// PLC -> Robot 外圍設備Input(Fanuc Robot的外圍)
MEMMOVE(
destAddr:=ADR(_rawOut_UO[0])
,srcAddr:=ADR(_UI1)
,n:=4
);
// PLC -> Robot Digital Output 2byte(send the command to Fanuc Robot), Warehouse Robot move ClampA
MEMMOVE(
destAddr:=ADR(_rawOut_DO[0])
,srcAddr:=ADR(_DO1)
,n:=2 
);
// PLC -> Robot Digital Output 2byte(send the command to Fanuc Robot), Warehouse Robot move ClampB
MEMMOVE(
destAddr:=ADR(_rawOut_DO[2])
,srcAddr:=ADR(_DO2)
,n:=2 
);
// PLC -> Robot Digital Output 2byte(send the command to Fanuc Robot), ABS Robot move ClampA
MEMMOVE(
destAddr:=ADR(_rawOut_DO[4])
,srcAddr:=ADR(_DO3)
,n:=2 
);
// PLC -> Robot Digital Output 2byte(send the command to Fanuc Robot), ABS Robot move ClampA
MEMMOVE(
destAddr:=ADR(_rawOut_DO[6])
,srcAddr:=ADR(_DO4)
,n:=2 
);
// PLC -> Robot Digital output 2byte(send the command to Fanuc Robot), General Command
MEMMOVE(
destAddr:=ADR(_rawOut_DO[8])
,srcAddr:=ADR(_DO5)
,n:=2 
);
MEMMOVE(
destAddr:=ADR(_rawOut_DO[10])
,srcAddr:=ADR(_DO6)
,n:=2 
);
MEMMOVE(
destAddr:=ADR(_rawOut_DO[12])
,srcAddr:=ADR(_DO7)
,n:=2 
);
MEMMOVE(
destAddr:=ADR(_rawOut_DO[14])
,srcAddr:=ADR(_DO8)
,n:=2 
);
MEMMOVE(
destAddr:=ADR(_rawOut_DO[16])
,srcAddr:=ADR(_DO9)
,n:=2 
);

MEMMOVE(
destAddr:=ADR(_rawOut_DO[18])
,srcAddr:=ADR(_DO10)
,n:=2 
);
MEMMOVE(
destAddr:=ADR(_rawOut_DO[20])
,srcAddr:=ADR(_DO11)
,n:=2 
);
MEMMOVE(
destAddr:=ADR(_rawOut_DO[22])
,srcAddr:=ADR(_DO12)
,n:=2 
);
MEMMOVE(
destAddr:=ADR(_rawOut_DO[24])
,srcAddr:=ADR(_DO13)
,n:=2 
);
MEMMOVE(
destAddr:=ADR(_rawOut_DO[26])
,srcAddr:=ADR(_DO14)
,n:=2 
);
MEMMOVE(
destAddr:=ADR(_rawOut_DO[28])
,srcAddr:=ADR(_DO15)
,n:=2 
);
MEMMOVE(
destAddr:=ADR(_rawOut_DO[30])
,srcAddr:=ADR(_DO16)
,n:=2 
);


// Robot -> PLC Digital Input 3byte(Send Robot Status to PLC), All service
MEMMOVE(
destAddr:=ADR(_DI1)
,srcAddr:=ADR(_rawIn_DI[0])
,n:=3
);

MEMMOVE(
destAddr:=ADR(_DI2)
,srcAddr:=ADR(_rawIn_DI[3])
,n:=2
);
MEMMOVE(
destAddr:=ADR(_DI3)
,srcAddr:=ADR(_rawIn_DI[5])
,n:=2
);
MEMMOVE(
destAddr:=ADR(_DI4)
,srcAddr:=ADR(_rawIn_DI[7])
,n:=2
);
MEMMOVE(
destAddr:=ADR(_DI5)
,srcAddr:=ADR(_rawIn_DI[9])
,n:=2
);
MEMMOVE(
destAddr:=ADR(_DI6)
,srcAddr:=ADR(_rawIn_DI[11])
,n:=2
);
MEMMOVE(
destAddr:=ADR(_DI7)
,srcAddr:=ADR(_rawIn_DI[13])
,n:=2
);
MEMMOVE(
destAddr:=ADR(_DI8)
,srcAddr:=ADR(_rawIn_DI[15])
,n:=2
);
MEMMOVE(
destAddr:=ADR(_DI9)
,srcAddr:=ADR(_rawIn_DI[17])
,n:=2
);
MEMMOVE(
destAddr:=ADR(_DI10)
,srcAddr:=ADR(_rawIn_DI[19])
,n:=2
);
MEMMOVE(
destAddr:=ADR(_DI11)
,srcAddr:=ADR(_rawIn_DI[21])
,n:=2
);
MEMMOVE(
destAddr:=ADR(_DI12)
,srcAddr:=ADR(_rawIn_DI[23])
,n:=2
);

// Robot Status com
qEnable:=_UO1.UO01_CmdEnabled AND _UO1.UO02_SystemReady;
Error:=Fault();

// Velocity Command transfer
_DO5.VelocityBit0 := _VelocityCommand.BitList.Bit0;
_DO5.VelocityBit1 := _VelocityCommand.BitList.Bit1;
_DO5.VelocityBit2 := _VelocityCommand.BitList.Bit2;
_DO5.VelocityBit3 := _VelocityCommand.BitList.Bit3;
_DO5.VelocityBit4 := _VelocityCommand.BitList.Bit4;
_DO5.VelocityBit5 := _VelocityCommand.BitList.Bit5;
_DO5.VelocityBit6 := _VelocityCommand.BitList.Bit6;
_DO5.VelocityBit7 := _VelocityCommand.BitList.Bit7;
END_METHOD

{attribute 'monitoring' := 'variable'}
PROPERTY VelocityCommand : Int
GET
VelocityCommand :=_VelocityCommand.nInt;
END_GET
SET
_VelocityCommand.nInt :=VelocityCommand;
END_SET
END_PROPERTY

PROPERTY WareHouseClampA_Handshake : ST_Fanuc_WarehouseHandshake
GET
WareHouseClampA_Handshake := _DO1;
END_GET
SET
// Outside -> FB 
_DO1 := WareHouseClampA_Handshake;
END_SET
END_PROPERTY

PROPERTY WareHouseClampB_Handshake : ST_Fanuc_WarehouseHandshake
GET
WareHouseClampB_Handshake := _DO2;
END_GET
SET
// Outside -> FB 
_DO2 := WareHouseClampB_Handshake;
END_SET
END_PROPERTY

PROPERTY Write_OffsetP : INT
SET
_DI11 := Write_OffsetP;
END_SET
END_PROPERTY

PROPERTY Write_OffsetR : INT
SET
_DO12 := Write_OffsetR;
END_SET
END_PROPERTY

PROPERTY Write_OffsetW : INT
SET
_DO10 := Write_OffsetW;
END_SET
END_PROPERTY

PROPERTY Write_OffsetX : INT
SET
_DO7 := Write_OffsetX;
END_SET
END_PROPERTY

PROPERTY Write_OffsetY : INT
SET
_DO8 := Write_OffsetY;
END_SET
END_PROPERTY

PROPERTY Write_OffsetZ : INT
SET
_DO9 := Write_OffsetZ;
END_SET
END_PROPERTY

PROPERTY WriteDataCommand : bool;
SET
_DO6.WritePara_Execute := WriteDataCommand;
END_SET
END_PROPERTY

END_FUNCTION_BLOCK

// ---- Library/20_MachineUnits/21_StorageArea/Old_version_Service/FB_FeedInEmptyBoxWithRobot.TcPOU
FUNCTION_BLOCK FB_FeedInEmptyBoxWithRobot EXTENDS FB_ObjectBase_V2 IMPLEMENTS IBasicElement
VAR_INPUT
    // Below are the components being controlled.
    Robot           : REFERENCE TO FB_FanucRobot_Basic_V2; // Fanuc Robot
    PullOutConveyor : REFERENCE TO FB_PullOutConveyorAction; // Allocated area pull out conveyor
    DiffSizeCV  : REFERENCE TO FB_Motor; // Allocated area feed in conveyor(diff and same size conveyor)
	SameSizeCV : REFERENCE TO FB_Motor;
    WareHouse       : REFERENCE TO FB_WareHouse; // Storage area warehouse A and warehouse B conveyor and sensor
    //SameSizeFullSensor : REFERENCE TO BOOL; 				 // Because the same size sensor implement FB_ConveyorSameSize, so use reference to connect it
    Info  : ST_FeedInEmptyBox_Info; // Setting the feedin emptybox action's parameter
    Input : REFERENCE TO ST_InputTable;
    Stop  : BOOL;
END_VAR
VAR_OUTPUT
END_VAR
VAR
    tonPlaceSensorDelay    : TON;
    tonFeedInConveyorDelay : TON;
    tonTimeOut             : TON;
    tonFeedBoxTimeout      : TON;
    strStatus              : STRING;
    _UniqueErrorCode       : STRING;
    _Abort                 : BOOL;
    uiResumeStep           : DINT;
    PreviousStrStatus      : STRING;
    PreviousErrorCode      : STRING;
	
	//2025/11/17 edit by Gamin
	TON_SameSizeCVmove	: TON;
	TON_DiffSizeCVmove	: TON;
END_VAR

SUPER^.A10_StateControl();
A00_BasicUnits();

ACTION A00_BasicUnits:
tonTimeOut(PT:=T#300S);
tonFeedBoxTimeout(PT:=T#15S);
tonPlaceSensorDelay(PT:=T#1S);
tonFeedInConveyorDelay(PT:=T#500MS);

//
TON_SameSizeCVmove(PT :=T#1S);
TON_DiffSizeCVmove(PT :=T#1S);
END_ACTION

METHOD M_CheckCommand : BOOL
VAR_INPUT
END_VAR

VAR_INST
	CheckBehavior : BOOL; // True : Behavior is correct
	CheckWareHouseSetting : BOOL; // True : WareHouse setting is correct
	CheckPullOutConveyorSetting : BOOL; // True : PullOut Conveyor setting is correct
	CheckPickUpArea : BOOL; // True : PickUp Area is correct
	CheckPlaceArea : BOOL; // True : Place Area is correct
END_VAR
// Memory clear
CheckBehavior := FALSE;
// Check command is correct
IF info.ClampA_Setting.Behavior = E_ClampWork.Work OR info.ClampB_Setting.Behavior = E_ClampWork.Work THEN
	CheckBehavior := TRUE;
ELSE
	CheckBehavior := FALSE;
END_IF


M_CheckCommand := CheckBehavior;
END_METHOD

METHOD M_CheckUnitsNotBusy : BOOL
VAR_INPUT
END_VAR
M_CheckUnitsNotBusy := true; // need add units check
END_METHOD

METHOD M_CheckUnitsReady : BOOL
VAR_INPUT
END_VAR
M_CheckUnitsReady := NOT (Robot.Error (*OR PullOutConveyor.Error OR FeedInConveyor.bError OR WareHouse.bError*));
END_METHOD

METHOD M_ReloadBox
VAR_INPUT
	Info : ST_FeedInEmptyBox_Info;
END_VAR
IF info.PickUpArea    = E_FeedInEmptyBox_PickUpArea.PullOutConveyorA THEN
    uiExecutingStep   := 1000;
ELSIF info.PickUpArea = E_FeedInEmptyBox_PickUpArea.PullOutConveyorB THEN
    uiExecutingStep   := 2000;
ELSIF info.PickUpArea = E_FeedInEmptyBox_PickUpArea.WareHouseA THEN
    //WareHouse.
ELSIF info.PickUpArea = E_FeedInEmptyBox_PickUpArea.WareHouseB THEN
    uiExecutingStep   := 4000;
ELSE
    _Error := TRUE;
    Status := 'PickUp area value is out of range';
END_IF
END_METHOD

METHOD M_ReloadPulloutConveyorBox : BOOL
VAR_INPUT
	Execute : BOOL;
	SlideSelect : E_PullOutConveyorPosition;
END_VAR
VAR_INST
	uiReloadPulloutConveyorBoxStep : UDINT;
	fbExecute_Rtrig : R_TRIG;
	fbExecute_Ftrig : F_TRIG;
END_VAR
fbExecute_Rtrig(CLK := Execute);
fbExecute_Ftrig(CLK := Execute);
IF fbExecute_Rtrig.Q THEN
	uiReloadPulloutConveyorBoxStep := 100;
ELSIF fbExecute_Ftrig.Q THEN
	uiReloadPulloutConveyorBoxStep := 99000;
END_IF
CASE uiReloadPulloutConveyorBoxStep OF
	0 : 
		// Wait command
	99000:
//		PullOutConveyor.FixCylinderA1.M_MoveBackward('');
//		PullOutConveyor.FixCylinderA2.M_MoveBackward('');
//		PullOutConveyor.FixCylinderB1.M_MoveBackward('');
//		PullOutConveyor.FixCylinderB2.M_MoveBackward('');
END_CASE
END_METHOD

METHOD M_SelectActionMode : E_FeedInAction
VAR_INPUT
END_VAR
IF info.ClampA_Setting.Behavior = E_ClampWork.Work AND info.ClampB_Setting.Behavior <> E_ClampWork.Work THEN
	IF info.ClampA_Setting.PickUpArea = E_FeedInEmptyBox_PickUpArea.WareHouseA THEN
		M_SelectActionMode := E_FeedInAction.ClampA_WareHouseA;
	ELSIF info.ClampA_Setting.PickUpArea = E_FeedInEmptyBox_PickUpArea.WareHouseB THEN
		M_SelectActionMode := E_FeedInAction.ClampA_WareHouseB;
	ELSIF info.ClampA_Setting.PickUpArea = E_FeedInEmptyBox_PickUpArea.PullOutConveyor THEN
		M_SelectActionMode := E_FeedInAction.ClampA_PullOutConveyor;
	END_IF
ELSIF info.ClampA_Setting.Behavior <> E_ClampWork.Work AND info.ClampB_Setting.Behavior = E_ClampWork.Work THEN
	IF info.ClampB_Setting.PickUpArea = E_FeedInEmptyBox_PickUpArea.WareHouseA THEN
		M_SelectActionMode := E_FeedInAction.ClampB_WareHouseA;
	ELSIF info.ClampB_Setting.PickUpArea = E_FeedInEmptyBox_PickUpArea.WareHouseB THEN
		M_SelectActionMode := E_FeedInAction.ClampB_WareHouseB;
	ELSIF info.ClampB_Setting.PickUpArea = E_FeedInEmptyBox_PickUpArea.PullOutConveyor THEN
		M_SelectActionMode := E_FeedInAction.ClampB_PullOutConveyor;
	END_IF
ELSIF info.ClampA_Setting.Behavior = E_ClampWork.Work AND info.ClampB_Setting.Behavior = E_ClampWork.Work THEN
	IF info.ClampA_Setting.PickUpArea = E_FeedInEmptyBox_PickUpArea.PullOutConveyor THEN
		IF  info.ClampB_Setting.PickUpArea = E_FeedInEmptyBox_PickUpArea.WareHouseA THEN
			M_SelectActionMode := E_FeedInAction.A_PullOut_B_WareHouseA;
		ELSIF info.ClampB_Setting.PickUpArea = E_FeedInEmptyBox_PickUpArea.WareHouseB THEN
			M_SelectActionMode := E_FeedInAction.A_PullOut_B_WareHouseB;
		ELSIF info.ClampB_Setting.PickUpArea = E_FeedInEmptyBox_PickUpArea.PullOutConveyor THEN
			M_SelectActionMode := E_FeedInAction.A_PullOut_B_PullOut;
		END_IF
	ELSIF info.ClampA_Setting.PickUpArea = E_FeedInEmptyBox_PickUpArea.WareHouseA THEN
		IF info.ClampB_Setting.PickUpArea = E_FeedInEmptyBox_PickUpArea.WareHouseA THEN
			M_SelectActionMode := E_FeedInAction.A_WareHouseA_B_WareHouseA;
		ELSIF info.ClampB_Setting.PickUpArea = E_FeedInEmptyBox_PickUpArea.WareHouseB THEN
			M_SelectActionMode := E_FeedInAction.A_WareHouseA_B_WareHouseB;
		ELSIF info.ClampB_Setting.PickUpArea = E_FeedInEmptyBox_PickUpArea.PullOutConveyor THEN
			M_SelectActionMode := E_FeedInAction.A_WareHouseA_B_PullOut;
		END_IF
	ELSIF info.ClampA_Setting.PickUpArea = E_FeedInEmptyBox_PickUpArea.WareHouseB THEN
		IF info.ClampB_Setting.PickUpArea = E_FeedInEmptyBox_PickUpArea.WareHouseA THEN
			M_SelectActionMode := E_FeedInAction.A_WareHouseB_B_WareHouseA;
		ELSIF info.ClampB_Setting.PickUpArea = E_FeedInEmptyBox_PickUpArea.WareHouseB THEN
			M_SelectActionMode := E_FeedInAction.A_WareHouseB_B_WareHouseB;
		ELSIF info.ClampB_Setting.PickUpArea = E_FeedInEmptyBox_PickUpArea.PullOutConveyor THEN
			M_SelectActionMode := E_FeedInAction.A_WareHouseB_B_PullOut;
		END_IF
	END_IF
END_IF
END_METHOD

METHOD  M_STATE_ABORTED
VAR_INPUT
END_VAR
Busy    := FALSE;
Aborted := TRUE;
Status := strStatus ;
UniqueErrorCode := _UniqueErrorCode;
IF NOT Execute THEN
    eState := STATE_RESETTING;
END_IF

IF Execute AND Reset THEN
	uiExecutingStep :=uiResumeStep;
	PreviousStrStatus := strStatus;
	PreviousErrorCode := _UniqueErrorCode;
	eState :=STATE_EXECUTING;
END_IF
END_METHOD

METHOD  M_STATE_ABORTING
VAR_INPUT
END_VAR
_AbortCompleted := TRUE;
_Abort :=FALSE;
tonTimeOut.IN:=FALSE;
//DAS.fbStorageArea.M_ResetSlideA_FeedIn();
IF strStatus = PreviousStrStatus THEN
	_UniqueErrorCode :=PreviousErrorCode;
END_IF
IF _AbortCompleted THEN
    eState := STATE_Aborted;
END_IF
END_METHOD

METHOD  M_STATE_DONE
VAR_INPUT
END_VAR
Busy := FALSE;
Done := TRUE;
IF NOT Execute THEN
    eState := STATE_RESETTING;
END_IF
END_METHOD

METHOD  M_STATE_DORMANT
VAR_INPUT
END_VAR
// Clear FB output
Busy            := FALSE;
Done            := FALSE;
Aborted         := FALSE;
Error           :=  FALSE;
ErrorID         := 0;
Status          := '';
_ResetCompleted := FALSE;
_Error          := FALSE;
_Executed       := FALSE;
uiExecutingStep := 0;
uiResettingStep := 0;
uiResumeStep:=0;
tonPlaceSensorDelay.IN :=FALSE;
tonFeedInConveyorDelay.IN :=FALSE;
tonTimeOut.IN :=FALSE;
TON_DiffSizeCVmove.IN := FALSE;
TON_SameSizeCVmove.IN := FALSE;
_UniqueErrorCode :='0';
PreviousStrStatus			 :='';
PreviousErrorCode			 :='';
//DAS.fbStorageArea.M_InactivePulloutConveyorInternCtrl();
// Wait Execute command
IF Execute THEN
    eState := STATE_EXECUTING;
END_IF
END_METHOD

METHOD  M_STATE_ERROR
VAR_INPUT
END_VAR
Robot.Bzone_AllowWork:=FALSE;
IF NOT Execute THEN
    eState := STATE_RESETTING;
END_IF
END_METHOD

METHOD M_STATE_EXECUTING
VAR_INPUT
END_VAR
VAR_INST
    ClampA_WareHouseCoordinates : ST_WareHouseCoordinates;
    ClampB_WareHouseCoordinates : ST_WareHouseCoordinates;
    uiPickUpBothStep            : UINT;
    uiPlaceBothStep             : UINT;
    BoxReady_1st                : BOOL;
    BoxReady_2nd                : BOOL;
    SlideClear_1st              : BOOL;
    SlideClear_2nd              : BOOL;
    TargetWarehouse             : E_WareHouse;
    DiffSizeSlide_Clear         : BOOL;
    SameSizeSlide_clear         : BOOL;
    ActionMode                  : E_FeedInAction;
END_VAR
VAR

END_VAR
// Set status busy
Busy := TRUE;
Robot.Bzone_AllowWork:=Robot._DI12.BzoneInWork;
//Auto mode , just allow robot
IF THIS^.Stop THEN // Pending the timeout when Stop signal occur
  tonTimeout.IN :=FALSE;
END_IF
CASE uiExecutingStep OF
    0:
        // Clear variable
        ActionMode       := E_FeedInAction.Undefined;
        BoxReady_1st     := FALSE;
        BoxReady_2nd     := FALSE;
        uiPickUpBothStep := 0;
        uiPlaceBothStep  := 0;

        // Check command
        IF M_CheckCommand() THEN
            uiExecutingStep := 10;
        END_IF
    10: // Start process, check units first
        IF M_CheckUnitsReady() THEN
            uiExecutingStep := 20;
        END_IF
    20: // Check units not busy state
        IF M_CheckUnitsNotBusy() THEN
            uiExecutingStep := 1000;
        END_IF
    1000:
        // Select action mode
        ActionMode      := M_SelectActionMode();
        uiExecutingStep := 1100;
    1100:
        // according action mode jump step
        CASE ActionMode OF
            E_FeedInAction.ClampA_WareHouseA:
                uiExecutingStep := 10000; // Go to start only ClampA pickup from WareHouseA
            E_FeedInAction.ClampA_WareHouseB:
                uiExecutingStep := 11000; // Go to Start only ClampA pickup from WareHouseB
            E_FeedInAction.ClampA_PullOutConveyor:
                uiExecutingStep := 12000; // Go to Start only ClampA pickup form PulloutConveyor
            E_FeedInAction.ClampB_WareHouseA:
                uiExecutingStep := 20000; // Go to Start only ClampB pickup from WareHouseA
            E_FeedInAction.ClampB_WareHouseB:
                uiExecutingStep := 21000; // Go to Start only ClampB pickup from WareHouseB
            E_FeedInAction.ClampB_PullOutConveyor:
                uiExecutingStep := 22000; // Go to Start only ClampB pickup from PulloutConveyor
            E_FeedInAction.A_WareHouseA_B_WareHouseA:
                uiExecutingStep := 30000; // Go to Start ClampA pickup from WarehouseA, ClampB pickup from WarehouseA
            E_FeedInAction.A_WareHouseA_B_WareHouseB:
                uiExecutingStep := 31000; // Go to Start ClampA pickup from WarehouseA, ClmapB pickup from WarehouseB
            E_FeedInAction.A_WareHouseA_B_PullOut:
                uiExecutingStep := 32000; // Go to Start ClampA pickup from WarehouseA, ClampB pickup from PulloutConveyor
            E_FeedInAction.A_WareHouseB_B_WareHouseA:
                uiExecutingStep := 33000; // Go to Start ClampA pickup from WarehouseB, ClampB pickup from WarehouseA
            E_FeedInAction.A_WareHouseB_B_WareHouseB:
                uiExecutingStep := 34000; // Go to Start ClampA pickup from WarehouseB, CLampB pickup from WarehouseB
            E_FeedInAction.A_WareHouseB_B_PullOut:
                uiExecutingStep := 35000; // Go to Start ClampA pickup from WarehouseB, ClampB pickup from PulloutConveyor
            E_FeedInAction.A_PullOut_B_WareHouseA:
                uiExecutingStep := 36000; // Go to Start ClampA pickup from PulloutConveyor, ClampB pickup from WarehouseA
            E_FeedInAction.A_PullOut_B_WareHouseB:
                uiExecutingStep := 37000; // Go to Start ClampA pickup from PulloutConveyor, ClampB pickup from WarehouseB
            E_FeedInAction.A_PullOut_B_PullOut:
                uiExecutingStep := 38000; // Go to Start ClampBoth pickup from PulloutConveyor
        END_CASE
    10000: // Only clampA pickup box from WareHouseA
        IF NOT Robot._DI1.Done THEN
            ClampA_WareHouseCoordinates := info.ClampA_Setting.WareHouseSetting;
            WareHouse.M_StartReloadBox(WareHouseSelect := E_WareHouse.WareHouseA, WarehouseCoordinates := ClampA_WareHouseCoordinates);

            IF WareHouse.bReloadBox_Completed THEN
                BoxReady_1st := TRUE;
            END_IF

            Robot.M_StartWareHousePickUpBox_ClampA(WareHouseSelect := E_WareHouse.WareHouseA,
                                                   Info            := ClampA_WareHouseCoordinates,
                                                   BoxReady_1st    := BoxReady_1st);
        ELSE
            IF Robot.M_ResetWareHousePickUpBox_ClampA() THEN
                // Clear command and go to place box
        tonTimeOut.IN:=FALSE;
                uiExecutingStep := 60000; // only place clampA
            END_IF
        END_IF
    tonTimeOut.IN :=TRUE;   
    IF tonTimeOut.Q THEN
      tonTimeOut.IN:=FALSE;
      _Error :=TRUE;
      strStatus :='Pick Box timeout';
    END_IF
    
    11000: // Only ClampA pickup box from WareHouseB
        IF NOT Robot._di1.Done THEN
            ClampA_WareHouseCoordinates := info.ClampA_Setting.WareHouseSetting;
            WareHouse.M_StartReloadBox(WareHouseSelect := E_WareHouse.WareHouseB, WarehouseCoordinates := ClampA_WareHouseCoordinates);

            IF WareHouse.bReloadBox_Completed THEN
                BoxReady_1st := TRUE;
            END_IF

            Robot.M_StartWareHousePickUpBox_ClampA(WareHouseSelect := E_WareHouse.WareHouseB,
                                                   Info            := ClampA_WareHouseCoordinates,
                                                   BoxReady_1st    := BoxReady_1st);
        ELSE
            IF Robot.M_ResetWareHousePickUpBox_ClampA() THEN
                // Clear command and go to place box
        tonTimeOut.IN:=FALSE;
                uiExecutingStep := 60000; // only place clampA
            END_IF
        END_IF

    tonTimeOut.IN :=TRUE;   
    IF tonTimeOut.Q THEN
      tonTimeOut.IN:=FALSE;
      _Error :=TRUE;
      strStatus :='Pick Box timeout';
    END_IF
    
    12000: // Only ClampA pickup box from pullout conveyor
        IF NOT Robot._di1.Done THEN
            DAS_CoreSys.MachineControl.fbStorageArea.M_ActivePulloutConveyorInternCtrl();

            IF Info.ClampA_Setting.PullOutConveyorSetting = E_PullOutConveyorAddress.I3_Slide THEN
                DAS_CoreSys.MachineControl.fbStorageArea.M_StartSlideB_FeedIn();
            ELSIF Info.ClampA_Setting.PullOutConveyorSetting = E_PullOutConveyorAddress.I4_Slide THEN
                DAS_CoreSys.MachineControl.fbStorageArea.M_StartSlideA_FeedIn();
            ELSE
                Status := 'Not define PulloutConveyor Slide';
                _Error := TRUE;
            END_IF

            Robot.M_StartPullOutConveyorPickUpBox_ClampA(ClampA_Address := Info.ClampA_Setting.PullOutConveyorSetting,
                                                         BoxReady       := DAS_CoreSys.MachineControl.fballocatearea.fbPulloutCV.Done);
        ELSE
            IF Robot.M_ResetPullOutConveyorPickUpBox_ClampA() THEN
                DAS_CoreSys.MachineControl.fbStorageArea.M_ResetSlideA_FeedIn();
        tonTimeOut.IN:=FALSE;
                uiExecutingStep := 60000; // only place clampA
            END_IF
        END_IF;
      tonTimeOut.IN :=TRUE;   
    IF tonTimeOut.Q THEN
      tonTimeOut.IN:=FALSE;
      _Abort :=TRUE;
      uiResumeStep:=12000;
      strStatus :='Pick Box timeout';
    END_IF
    
    20000: // Only clampB pickup box from WareHouseA
        IF NOT Robot._di1.Done THEN
            ClampB_WareHouseCoordinates := info.ClampB_Setting.WareHouseSetting;
            WareHouse.M_StartReloadBox(WareHouseSelect := E_WareHouse.WareHouseA, WarehouseCoordinates := ClampB_WareHouseCoordinates);

            IF WareHouse.bReloadBox_Completed THEN
                BoxReady_2nd := TRUE;
            END_IF

            Robot.M_StartWareHousePickUpBox_ClampB(WareHouseSelect := E_WareHouse.WareHouseA,
                                                   Info            := ClampB_WareHouseCoordinates,
                                                   BoxReady_2nd    := BoxReady_2nd);
        ELSE
            IF Robot.M_ResetWareHousePickUpBox_ClampB() THEN
                // Clear command and go to place box
        tonTimeOut.IN:=FALSE;
                uiExecutingStep := 70000; // only place clampA
            END_IF
        END_IF
      tonTimeOut.IN :=TRUE;   
    IF tonTimeOut.Q THEN
      tonTimeOut.IN:=FALSE;
      _Error :=TRUE;
      strStatus :='Pick Box timeout';
    END_IF
    21000: // Only ClampB pickup box from WareHouseB
        IF NOT Robot._di1.Done THEN
            ClampB_WareHouseCoordinates := info.ClampB_Setting.WareHouseSetting;
            WareHouse.M_StartReloadBox(WareHouseSelect := E_WareHouse.WareHouseB, WarehouseCoordinates := ClampB_WareHouseCoordinates);

            IF WareHouse.bReloadBox_Completed THEN
                BoxReady_2nd := TRUE;
            END_IF

            Robot.M_StartWareHousePickUpBox_ClampB(WareHouseSelect := E_WareHouse.WareHouseB,
                                                   Info            := ClampB_WareHouseCoordinates,
                                                   BoxReady_2nd    := BoxReady_2nd);
        ELSE
            IF Robot.M_ResetWareHousePickUpBox_ClampB() THEN
                // Clear command and go to place box
        tonTimeOut.IN:=FALSE;
                uiExecutingStep := 70000; // only place clampA
            END_IF
        END_IF
        tonTimeOut.IN :=TRUE;   
    IF tonTimeOut.Q THEN
      tonTimeOut.IN:=FALSE;
      _Error :=TRUE;
      strStatus :='Pick Box timeout';
    END_IF

    22000: // Only ClampB pickup box from PullOut conveyor
        IF NOT Robot._di1.Done THEN
            DAS_CoreSys.MachineControl.fbStorageArea.M_ActivePulloutConveyorInternCtrl();

            IF Info.ClampB_Setting.PullOutConveyorSetting = E_PullOutConveyorAddress.I3_Slide THEN
                DAS_CoreSys.MachineControl.fbStorageArea.M_StartSlideB_FeedIn();
            ELSIF Info.ClampB_Setting.PullOutConveyorSetting = E_PullOutConveyorAddress.I4_Slide THEN
                DAS_CoreSys.MachineControl.fbStorageArea.M_StartSlideA_FeedIn();
            ELSE
                Status := 'Not define PulloutConveyor Slide';
                _Error := TRUE;
            END_IF

            Robot.M_StartPullOutConveyorPickUpBox_ClampB(ClampB_Address := Info.ClampB_Setting.PullOutConveyorSetting,
                                                         BoxReady       := DAS_CoreSys.MachineControl.fballocatearea.fbPulloutCV.Done);
        ELSE
            IF Robot.M_ResetPullOutConveyorPickUpBox_ClampB() THEN
                DAS_CoreSys.MachineControl.fbStorageArea.M_ResetSlideA_FeedIn();
        tonTimeOut.IN:=FALSE;
                uiExecutingStep := 70000; // only place clampA
            END_IF
        END_IF;
      tonTimeOut.IN :=TRUE;   
    IF tonTimeOut.Q THEN
      uiResumeStep:=22000;
      _Abort :=TRUE;
      strStatus :='Pick Box timeout';
    END_IF
    
    30000: // ClampA pickup from WarehouseA, ClampB pickup from WarehouseA
        ClampA_WareHouseCoordinates := info.ClampA_Setting.WareHouseSetting;
        ClampB_WareHouseCoordinates := info.ClampB_Setting.WareHouseSetting;

        CASE uiPickUpBothStep OF
            0: // ClampA target slide move the box to front side
                WareHouse.M_StartReloadBox(WareHouseSelect := E_WareHouse.WareHouseA, WarehouseCoordinates := ClampA_WareHouseCoordinates);

                IF WareHouse.bReloadBox_Completed THEN
                    BoxReady_1st     := TRUE;
                    uiPickUpBothStep := 10;
                END_IF

            10: // wait Robot Allow continue
                IF Robot._DI1.Notification AND
                    NOT
                    WareHouse._stWarehouseList.ASide_Layers[ClampA_WareHouseCoordinates.Layer].stStatus.bSlides[ClampA_WareHouseCoordinates.Slide]
                    THEN
                    WareHouse.M_ResetReloadBox();

                    IF NOT WareHouse.bReloadBox_Completed THEN
                        uiPickUpBothStep := 20;
                    END_IF

                END_IF
            20: // ClampB target slide move the box to front slide
                WareHouse.M_StartReloadBox(WareHouseSelect := E_WareHouse.WareHouseA, WarehouseCoordinates := ClampB_WareHouseCoordinates);

                IF WareHouse.bReloadBox_Completed THEN
                    BoxReady_2nd     := TRUE;
                    uiPickUpBothStep := 99;
                END_IF
            99:
        // wait reset
        END_CASE

        Robot.M_StartWareHousePickUpBox_ClampBoth(WareHouseSelect := E_WareHouse.WareHouseA,
                                                  ClampA_Info     := ClampA_WareHouseCoordinates,
                                                  ClampB_Info     := ClampB_WareHouseCoordinates,
                                                  BoxReady_1st    := BoxReady_1st,
                                                  BoxReady_2nd    := BoxReady_2nd);

        IF Robot._DI1.Done THEN
      tonTimeOut.IN:=FALSE;
            uiExecutingStep := 80000; // go to place step
        END_IF
      tonTimeOut.IN :=TRUE;   
    IF tonTimeOut.Q THEN
      tonTimeOut.IN:=FALSE;
      _Error :=TRUE;
      strStatus :='Pick Box timeout';
    END_IF
    
    31000: // ClampA pickup from WarehouseA, ClampB pickup from WarehouseB
        IF NOT Robot._DI1.Done THEN
            ClampA_WareHouseCoordinates := info.ClampA_Setting.WareHouseSetting;
            WareHouse.M_StartReloadBox(WareHouseSelect := E_WareHouse.WareHouseA, WarehouseCoordinates := ClampA_WareHouseCoordinates);

            IF WareHouse.bReloadBox_Completed THEN
                BoxReady_1st := TRUE;
            END_IF

            Robot.M_StartWareHousePickUpBox_ClampA(WareHouseSelect := E_WareHouse.WareHouseA,
                                                   Info            := ClampA_WareHouseCoordinates,
                                                   BoxReady_1st    := BoxReady_1st);
        ELSE
      tonTimeOut.IN:=FALSE;
      uiExecutingStep := 31080;
    END_IF
      tonTimeOut.IN :=TRUE;   
    IF tonTimeOut.Q THEN
      tonTimeOut.IN:=FALSE;
      _Error :=TRUE;
      strStatus :='Pick Box timeout';
    END_IF
    
  31080:
    Robot.M_ResetAllCommand(); // Clear command and go to place box
    IF NOT Robot._di1.Done THEN
      uiExecutingStep := 31100;// ClampA pickup finished, ClampB pickup start
    END_IF
    
    31100:
        IF NOT Robot._di1.Done THEN
            ClampB_WareHouseCoordinates := info.ClampB_Setting.WareHouseSetting;
            WareHouse.M_StartReloadBox(WareHouseSelect := E_WareHouse.WareHouseB, WarehouseCoordinates := ClampB_WareHouseCoordinates);

            IF WareHouse.bReloadBox_Completed THEN
                BoxReady_2nd := TRUE;
            END_IF

            Robot.M_StartWareHousePickUpBox_ClampB(WareHouseSelect := E_WareHouse.WareHouseB,
                                                   Info            := ClampB_WareHouseCoordinates,
                                                   BoxReady_2nd    := BoxReady_2nd);
        ELSE
      tonTimeOut.IN:=FALSE;
      uiExecutingStep := 31180;
    END_IF
      tonTimeOut.IN :=TRUE;   
    IF tonTimeOut.Q THEN
      tonTimeOut.IN:=FALSE;
      _Error :=TRUE;
      strStatus :='Pick Box timeout';
    END_IF
    
  31180:
    Robot.M_ResetAllCommand(); // Clear command and go to place box
    IF NOT Robot._di1.Done THEN
      uiExecutingStep := 80000;// ClampA pickup finished, ClampB pickup start
    END_IF
    32000: // ClampA pickup from WarehouseA, ClampB pickup from PulloutConveyor
        IF NOT Robot._DI1.Done THEN
            ClampA_WareHouseCoordinates := info.ClampA_Setting.WareHouseSetting;
            WareHouse.M_StartReloadBox(WareHouseSelect := E_WareHouse.WareHouseA, WarehouseCoordinates := ClampA_WareHouseCoordinates);

            IF WareHouse.bReloadBox_Completed THEN
                BoxReady_1st := TRUE;
            END_IF

            Robot.M_StartWareHousePickUpBox_ClampA(WareHouseSelect := E_WareHouse.WareHouseA,
                                                   Info            := ClampA_WareHouseCoordinates,
                                                   BoxReady_1st    := BoxReady_1st);
        ELSE
      tonTimeOut.IN:=FALSE;
      uiExecutingStep := 32080; // ClampA pickup finished, ClampB start 
        END_IF
      tonTimeOut.IN :=TRUE;   
    IF tonTimeOut.Q THEN
      tonTimeOut.IN:=FALSE;
      _Error :=TRUE;
      strStatus :='Pick Box timeout';
    END_IF
  32080:
    Robot.M_ResetAllCommand();
    // Clear command and go to place box
    IF NOT Robot._di1.Done THEN
      uiExecutingStep := 32100;// ClampA pickup finished, ClampB start
    END_IF
    32100:
        IF NOT Robot._di1.Done THEN
        DAS_CoreSys.MachineControl.fballocatearea.M_GetPulloutAccess(ControlAccess := E_RoundBeltControlAccess.FanucRobot);

            IF Info.ClampB_Setting.PullOutConveyorSetting = E_PullOutConveyorAddress.I3_Slide THEN
                        DAS_CoreSys.MachineControl.fballocatearea
                            .M_StartStoragePulloutAction(CommandType := E_PullOutConveyorCommandType.SlideB_FeedIn_Ext,
                                                         CV_BackwardTIme := T#0S,
                                                         CV_ForwardTime := T#0S);
            ELSIF Info.ClampB_Setting.PullOutConveyorSetting = E_PullOutConveyorAddress.I4_Slide THEN
                        DAS_CoreSys.MachineControl.fballocatearea
                            .M_StartStoragePulloutAction(CommandType := E_PullOutConveyorCommandType.SlideA_FeedIn_Ext,
                                                         CV_BackwardTIme := T#0S,
                                                         CV_ForwardTime := T#0S);
            ELSE
                Status := 'Not define PulloutConveyor Slide';
                _Error := TRUE;
            END_IF

            Robot.M_StartPullOutConveyorPickUpBox_ClampB(ClampB_Address := Info.ClampB_Setting.PullOutConveyorSetting,
                                                         BoxReady       := DAS_CoreSys.MachineControl.fballocatearea.fbPulloutCV.Done);
        ELSE
      tonTimeOut.IN:=FALSE;
      uiExecutingStep := 32180;
    END_IF
      tonTimeOut.IN :=TRUE;   
    IF tonTimeOut.Q THEN
      tonTimeOut.IN:=FALSE;
      _Error :=TRUE;
      strStatus :='Pick Box timeout';
    END_IF
  32180:
    robot.M_ResetAllCommand();
    IF NOT Robot._DI1.Done THEN
      uiExecutingStep := 80000;
    END_IF
    33000: // ClampA Pickup from WarehouseB, ClampB pickup from WarehouseA
        IF NOT Robot._di1.Done THEN
            ClampA_WareHouseCoordinates := info.ClampA_Setting.WareHouseSetting;
            WareHouse.M_StartReloadBox(WareHouseSelect := E_WareHouse.WareHouseB, WarehouseCoordinates := ClampA_WareHouseCoordinates);

            IF WareHouse.bReloadBox_Completed THEN
                BoxReady_1st := TRUE;
            END_IF

            Robot.M_StartWareHousePickUpBox_ClampA(WareHouseSelect := E_WareHouse.WareHouseB,
                                                   Info            := ClampA_WareHouseCoordinates,
                                                   BoxReady_1st    := BoxReady_1st);
        ELSE
      tonTimeOut.IN:=FALSE;
      uiExecutingStep := 33080;
    END_IF
        tonTimeOut.IN :=TRUE;   
    IF tonTimeOut.Q THEN
      tonTimeOut.IN:=FALSE;
      _Error :=TRUE;
      strStatus :='Pick Box timeout';
    END_IF
  33080:
    Robot.M_ResetAllCommand(); // Clear command and go to place box
    IF NOT Robot._DI1.Done THEN
                uiExecutingStep := 33100; // only place clampA
        END_IF
    33100:
        IF NOT Robot._di1.Done THEN
            ClampB_WareHouseCoordinates := info.ClampB_Setting.WareHouseSetting;
            WareHouse.M_StartReloadBox(WareHouseSelect := E_WareHouse.WareHouseA, WarehouseCoordinates := ClampB_WareHouseCoordinates);

            IF WareHouse.bReloadBox_Completed THEN
                BoxReady_2nd := TRUE;
            END_IF

            Robot.M_StartWareHousePickUpBox_ClampB(WareHouseSelect := E_WareHouse.WareHouseA,
                                                   Info            := ClampB_WareHouseCoordinates,
                                                   BoxReady_2nd    := BoxReady_2nd);
        ELSE
      Robot.M_ResetAllCommand(); // Clear command and go to place box
      IF NOT Robot._DI1.Done THEN
        tonTimeOut.IN:=FALSE;
        uiExecutingStep := 80000; // only place clampA
      END_IF
        END_IF
    tonTimeOut.IN :=TRUE;   
    IF tonTimeOut.Q THEN
      tonTimeOut.IN:=FALSE;
      _Error :=TRUE;
      strStatus :='Place Box timeout';
    END_IF
    
    34000: // ClampA pickup from WarehouseB, ClampB pickup from WarehouseB
        ClampA_WareHouseCoordinates := info.ClampA_Setting.WareHouseSetting;
        ClampB_WareHouseCoordinates := info.ClampB_Setting.WareHouseSetting;

        CASE uiPickUpBothStep OF
            0: // ClampA target slide move the box to front side
                WareHouse.M_StartReloadBox(WareHouseSelect := E_WareHouse.WareHouseB, WarehouseCoordinates := ClampA_WareHouseCoordinates);

                IF WareHouse.bReloadBox_Completed THEN
                    BoxReady_1st     := TRUE;
                    uiPickUpBothStep := 10;
                END_IF

            10: // wait Robot Allow continue
                IF Robot._DI1.Notification AND
                    NOT
                    WareHouse._stWarehouseList.BSide_Layers[ClampA_WareHouseCoordinates.Layer].stStatus.bSlides[ClampA_WareHouseCoordinates.Slide]
                    THEN
                    WareHouse.M_ResetReloadBox();

                    IF NOT WareHouse.bReloadBox_Completed THEN
                        uiPickUpBothStep := 20;
                    END_IF

                END_IF
            20: // ClampB target slide move the box to front slide
                WareHouse.M_StartReloadBox(WareHouseSelect := E_WareHouse.WareHouseB, WarehouseCoordinates := ClampB_WareHouseCoordinates);

                IF WareHouse.bReloadBox_Completed THEN
                    BoxReady_2nd     := TRUE;
                    uiPickUpBothStep := 99;
                END_IF
            99:
        // wait reset
        END_CASE

        Robot.M_StartWareHousePickUpBox_ClampBoth(WareHouseSelect := E_WareHouse.WareHouseB,
                                                  ClampA_Info     := ClampA_WareHouseCoordinates,
                                                  ClampB_Info     := ClampB_WareHouseCoordinates,
                                                  BoxReady_1st    := BoxReady_1st,
                                                  BoxReady_2nd    := BoxReady_2nd);

        IF Robot._DI1.Done THEN
      tonTimeOut.IN:=FALSE;
            uiExecutingStep := 80000; // go to place step
        END_IF
    
      tonTimeOut.IN :=TRUE;   
    IF tonTimeOut.Q THEN
      tonTimeOut.IN:=FALSE;
      _Error :=TRUE;
      strStatus :='Pick Box timeout';
    END_IF
    
    35000: // ClampA pickup from WarehouseB, ClampB pickup from PulloutConveyor
        IF NOT Robot._di1.Done THEN
        DAS_CoreSys.MachineControl.fballocatearea.M_GetPulloutAccess(ControlAccess := E_RoundBeltControlAccess.FanucRobot);

            IF Info.ClampA_Setting.PullOutConveyorSetting = E_PullOutConveyorAddress.I3_Slide THEN
                        DAS_CoreSys.MachineControl.fballocatearea
                            .M_StartStoragePulloutAction(CommandType := E_PullOutConveyorCommandType.SlideB_FeedIn_Ext,
                                                         CV_BackwardTIme := T#0S,
                                                         CV_ForwardTime := T#0S);
            ELSIF Info.ClampA_Setting.PullOutConveyorSetting = E_PullOutConveyorAddress.I4_Slide THEN
                        DAS_CoreSys.MachineControl.fballocatearea
                            .M_StartStoragePulloutAction(CommandType := E_PullOutConveyorCommandType.SlideA_FeedIn_Ext,
                                                         CV_BackwardTIme := T#0S,
                                                         CV_ForwardTime := T#0S);
            ELSE
                Status := 'Not define PulloutConveyor Slide';
                _Error := TRUE;
            END_IF

            Robot.M_StartPullOutConveyorPickUpBox_ClampA(ClampA_Address := Info.ClampA_Setting.PullOutConveyorSetting,
                                                         BoxReady       := DAS_CoreSys.MachineControl.fballocatearea.fbPulloutCV.Done);
        ELSE
            IF Robot.M_ResetPullOutConveyorPickUpBox_ClampA() THEN
            DAS_CoreSys.MachineControl.fballocatearea.M_StopStoragePulloutAction();
        tonTimeOut.IN:=FALSE;
                uiExecutingStep := 35100; // only place clampA
            END_IF
        END_IF;
      tonTimeOut.IN :=TRUE;   
    IF tonTimeOut.Q THEN
      tonTimeOut.IN:=FALSE;
      _Error :=TRUE;
      strStatus :='Pick Box timeout';
    END_IF
    
    35100:
        IF NOT Robot._di1.Done THEN
        DAS_CoreSys.MachineControl.fballocatearea.M_GetPulloutAccess(ControlAccess := E_RoundBeltControlAccess.FanucRobot);

            IF Info.ClampB_Setting.PullOutConveyorSetting = E_PullOutConveyorAddress.I3_Slide THEN
                        DAS_CoreSys.MachineControl.fballocatearea
                            .M_StartStoragePulloutAction(CommandType := E_PullOutConveyorCommandType.SlideB_FeedIn_Ext,
                                                         CV_BackwardTIme := T#0S,
                                                         CV_ForwardTime := T#0S);
            ELSIF Info.ClampB_Setting.PullOutConveyorSetting = E_PullOutConveyorAddress.I4_Slide THEN
                        DAS_CoreSys.MachineControl.fballocatearea
                            .M_StartStoragePulloutAction(CommandType := E_PullOutConveyorCommandType.SlideA_FeedIn_Ext,
                                                         CV_BackwardTIme := T#0S,
                                                         CV_ForwardTime := T#0S);
            ELSE
                Status := 'Not define PulloutConveyor Slide';
                _Error := TRUE;
            END_IF

            Robot.M_StartPullOutConveyorPickUpBox_ClampB(ClampB_Address := Info.ClampB_Setting.PullOutConveyorSetting,
                                                         BoxReady       := DAS_CoreSys.MachineControl.fballocatearea.fbPulloutCV.Done);
        ELSE
            IF Robot.M_ResetPullOutConveyorPickUpBox_ClampB() THEN
            DAS_CoreSys.MachineControl.fballocatearea.M_StopStoragePulloutAction();
        tonTimeOut.IN:=FALSE;
                uiExecutingStep := 80000; // only place clampA
            END_IF
        END_IF;
        tonTimeOut.IN :=TRUE;   
    IF tonTimeOut.Q THEN
      tonTimeOut.IN:=FALSE;
      _Error :=TRUE;
      strStatus :='Pick Box timeout';
    END_IF
    
    36000: // ClampA pickup from PulloutConveyor, ClampB pickup from WarehouseA
        IF NOT Robot._di1.Done THEN
        DAS_CoreSys.MachineControl.fballocatearea.M_GetPulloutAccess(ControlAccess := E_RoundBeltControlAccess.FanucRobot);

            IF Info.ClampA_Setting.PullOutConveyorSetting = E_PullOutConveyorAddress.I3_Slide THEN
                        DAS_CoreSys.MachineControl.fballocatearea
                            .M_StartStoragePulloutAction(CommandType := E_PullOutConveyorCommandType.SlideB_FeedIn_Ext,
                                                         CV_BackwardTIme := T#0S,
                                                         CV_ForwardTime := T#0S);
            ELSIF Info.ClampA_Setting.PullOutConveyorSetting = E_PullOutConveyorAddress.I4_Slide THEN
                        DAS_CoreSys.MachineControl.fballocatearea
                            .M_StartStoragePulloutAction(CommandType := E_PullOutConveyorCommandType.SlideA_FeedIn_Ext,
                                                         CV_BackwardTIme := T#0S,
                                                         CV_ForwardTime := T#0S);
            ELSE
                Status := 'Not define PulloutConveyor Slide';
                _Error := TRUE;
            END_IF

            Robot.M_StartPullOutConveyorPickUpBox_ClampA(ClampA_Address := Info.ClampA_Setting.PullOutConveyorSetting,
                                                         BoxReady       := DAS_CoreSys.MachineControl.fballocatearea.fbPulloutCV.Done);
        ELSE
      tonTimeOut.IN:=FALSE;
      uiExecutingStep := 36080;
    END_IF
        tonTimeOut.IN :=TRUE;   
    IF tonTimeOut.Q THEN
      tonTimeOut.IN:=FALSE;
      _Error :=TRUE;
      strStatus :='Pick Box timeout';
    END_IF
    
  36080:
    Robot.M_ResetAllCommand();
        DAS_CoreSys.MachineControl.fballocatearea.M_StopStoragePulloutAction();
    IF NOT Robot._di1.Done THEN
      uiExecutingStep := 36100; // only place clampA
    END_IF
    36100:
        IF NOT Robot._di1.Done THEN
            ClampB_WareHouseCoordinates := info.ClampB_Setting.WareHouseSetting;
            WareHouse.M_StartReloadBox(WareHouseSelect := E_WareHouse.WareHouseA, WarehouseCoordinates := ClampB_WareHouseCoordinates);

            IF WareHouse.bReloadBox_Completed THEN
                BoxReady_2nd := TRUE;
            END_IF

            Robot.M_StartWareHousePickUpBox_ClampB(WareHouseSelect := E_WareHouse.WareHouseA,
                                                   Info            := ClampB_WareHouseCoordinates,
                                                   BoxReady_2nd    := BoxReady_2nd);
        ELSE
      tonTimeOut.IN:=FALSE;
      uiExecutingStep := 36200;
    END_IF
        tonTimeOut.IN :=TRUE;   
    IF tonTimeOut.Q THEN
      tonTimeOut.IN:=FALSE;
      _Error :=TRUE;
      strStatus :='Pick Box timeout';
    END_IF
    
  36200:
    Robot.M_ResetAllCommand(); // Clear command and go to place box
    IF NOT Robot._DI1.Done THEN
      uiExecutingStep := 80000; //  place clampA and clampB
    END_IF 
    37000: // ClampA pickup from PulloutConveyor, ClampB pickup from WarehouseB
        IF NOT Robot._di1.Done THEN
        DAS_CoreSys.MachineControl.fballocatearea.M_GetPulloutAccess(ControlAccess := E_RoundBeltControlAccess.FanucRobot);

            IF Info.ClampA_Setting.PullOutConveyorSetting = E_PullOutConveyorAddress.I3_Slide THEN
                        DAS_CoreSys.MachineControl.fballocatearea
                            .M_StartStoragePulloutAction(CommandType := E_PullOutConveyorCommandType.SlideB_FeedIn_Ext,
                                                         CV_BackwardTIme := T#0S,
                                                         CV_ForwardTime := T#0S);
            ELSIF Info.ClampA_Setting.PullOutConveyorSetting = E_PullOutConveyorAddress.I4_Slide THEN
                        DAS_CoreSys.MachineControl.fballocatearea
                            .M_StartStoragePulloutAction(CommandType := E_PullOutConveyorCommandType.SlideA_FeedIn_Ext,
                                                         CV_BackwardTIme := T#0S,
                                                         CV_ForwardTime := T#0S);
            ELSE
                Status := 'Not define PulloutConveyor Slide';
                _Error := TRUE;
            END_IF

            Robot.M_StartPullOutConveyorPickUpBox_ClampA(ClampA_Address := Info.ClampA_Setting.PullOutConveyorSetting,
                                                         BoxReady       := DAS_CoreSys.MachineControl.fballocatearea.fbPulloutCV.Done);
        ELSE
      tonTimeOut.IN:=FALSE;
      uiExecutingStep := 37080;
    END_IF
          tonTimeOut.IN :=TRUE;   
    IF tonTimeOut.Q THEN
      tonTimeOut.IN:=FALSE;
      _Error :=TRUE;
      strStatus :='Pick Box timeout';
    END_IF
    
    
  37080:
    Robot.M_ResetAllCommand();
    IF NOT Robot._di1.Done THEN
      // Clear Pullout conveyor reload command
            DAS_CoreSys.MachineControl.fballocatearea.M_StopStoragePulloutAction();
      uiExecutingStep := 37100;
    END_IF
    37100:
        IF NOT Robot._di1.Done THEN
            ClampB_WareHouseCoordinates := info.ClampB_Setting.WareHouseSetting;
            WareHouse.M_StartReloadBox(WareHouseSelect := E_WareHouse.WareHouseB, WarehouseCoordinates := ClampB_WareHouseCoordinates);

            IF WareHouse.bReloadBox_Completed THEN
                BoxReady_2nd := TRUE;
            END_IF

            Robot.M_StartWareHousePickUpBox_ClampB(WareHouseSelect := E_WareHouse.WareHouseB,
                                                   Info            := ClampB_WareHouseCoordinates,
                                                   BoxReady_2nd    := BoxReady_2nd);
        ELSE
      tonTimeOut.IN:=FALSE;
      uiExecutingStep := 37180;
    END_IF
    tonTimeOut.IN :=TRUE;   
    IF tonTimeOut.Q THEN
      tonTimeOut.IN:=FALSE;
      _Error :=TRUE;
      strStatus :='Pick Box timeout';
    END_IF
  37180:
    Robot.M_ResetAllCommand(); // Clear command and go to place box
    IF NOT Robot._di1.Done THEN
      uiExecutingStep := 80000; // only place clampA
    END_IF
    38000: // ClampBoth pickup from PulloutConveyor
        DAS_CoreSys.MachineControl.fballocatearea.M_GetPulloutAccess(ControlAccess := E_RoundBeltControlAccess.FanucRobot);

        CASE uiPickUpBothStep OF
            0: // ClampA target slide move the box to front side
                IF Info.ClampA_Setting.PullOutConveyorSetting = E_PullOutConveyorAddress.I3_Slide THEN
                        DAS_CoreSys.MachineControl.fballocatearea
                            .M_StartStoragePulloutAction(CommandType := E_PullOutConveyorCommandType.SlideB_FeedIn_Ext,
                                                         CV_BackwardTIme := T#0S,
                                                         CV_ForwardTime := T#0S);
                ELSIF Info.ClampA_Setting.PullOutConveyorSetting = E_PullOutConveyorAddress.I4_Slide THEN
                        DAS_CoreSys.MachineControl.fballocatearea
                            .M_StartStoragePulloutAction(CommandType := E_PullOutConveyorCommandType.SlideA_FeedIn_Ext,
                                                         CV_BackwardTIme := T#0S,
                                                         CV_ForwardTime := T#0S);
                ELSE
                    Status := 'Not define PulloutConveyor Slide';
                    _Error := TRUE;
                END_IF

                IF DAS_CoreSys.MachineControl.fballocatearea.fbpulloutcv.Done THEN
                    BoxReady_1st     := TRUE;
                    uiPickUpBothStep := 10;
                END_IF

            10: // wait Robot Allow continue
                IF Robot._DI1.Notification THEN
                DAS_CoreSys.MachineControl.fballocatearea.M_StopStoragePulloutAction();

                    IF NOT DAS_CoreSys.MachineControl.fballocatearea.fbpulloutcv.Done THEN
                        uiPickUpBothStep := 20;
                    END_IF

                END_IF
            20: // ClampB target slide move the box to front slide
                IF Info.ClampB_Setting.PullOutConveyorSetting = E_PullOutConveyorAddress.I3_Slide THEN
                        DAS_CoreSys.MachineControl.fballocatearea
                            .M_StartStoragePulloutAction(CommandType := E_PullOutConveyorCommandType.SlideB_FeedIn_Ext,
                                                         CV_BackwardTIme := T#0S,
                                                         CV_ForwardTime := T#0S);
                ELSIF Info.ClampB_Setting.PullOutConveyorSetting = E_PullOutConveyorAddress.I4_Slide THEN
                        DAS_CoreSys.MachineControl.fballocatearea
                            .M_StartStoragePulloutAction(CommandType := E_PullOutConveyorCommandType.SlideA_FeedIn_Ext,
                                                         CV_BackwardTIme := T#0S,
                                                         CV_ForwardTime := T#0S);
                ELSE
                    Status := 'Not define PulloutConveyor Slide';
                    _Error := TRUE;
                END_IF

                IF DAS_CoreSys.MachineControl.fballocatearea.fbpulloutcv.Done THEN
                    BoxReady_2nd     := TRUE;
                    uiPickUpBothStep := 99;
                END_IF
            99:
        // wait reset
        END_CASE

        Robot.M_StartPullOutConveyorPickUpBox_ClampBoth(ClampA_Address := Info.ClampA_Setting.PullOutConveyorSetting,
                                                        ClampB_Address := Info.ClampB_Setting.PullOutConveyorSetting,
                                                        BoxReady_1     := BoxReady_1st,
                                                        BoxReady_2     := BoxReady_2nd);

        IF Robot._DI1.Done THEN
      tonTimeOut.IN:=FALSE;
            uiExecutingStep := 80000; // go to place step
        END_IF
    
    tonTimeOut.IN :=TRUE;   
    IF tonTimeOut.Q THEN
      tonTimeOut.IN:=FALSE;
      _Abort :=TRUE;  
      uiResumeStep:=38000;    
      strStatus :='Pick Box timeout';
    END_IF
    60000: // Only ClampA place box
        // Clear command
        WareHouse.M_ResetReloadBox();
        Robot.M_ResetAllCommand();

        // Check robot RSR1 not working
        IF NOT Robot._DI1.Done AND NOT (Robot._DI1.AbsMoveA OR Robot._DI1.AbsMoveB OR Robot._DI1.WarehouseA OR Robot._DI1.WarehouseB) THEN
            uiExecutingStep := 61000;
        END_IF
    61000: // Only ClampA place box Start
        IF NOT Robot._DI1.Done THEN
      IF NOT DiffSizeCV.InBackWard AND SameSizeCV.InBackWard THEN
        CASE Info.ClampA_Setting.PlaceArea OF
          E_FeedInEmptyBox_PlaceArea.DiffSizeConveyor:
          
                  DiffSizeCV.M_MoveForward();
          E_FeedInEmptyBox_PlaceArea.SameSizeConveyor:
            SameSizeCV.M_MoveForward();
        END_CASE

              IF Input.bDifferentSizeCV_BoxDetect7_Sensor THEN
                  DiffSizeSlide_Clear := FALSE;
              ELSE
                  DiffSizeSlide_Clear := TRUE;
              END_IF

              IF Input.bSameSizeCV_BoxNearStorageSensor THEN
                  SameSizeSlide_clear := FALSE;
              ELSE
                  SameSizeSlide_clear := TRUE;
              END_IF
      ELSE
          DiffSizeSlide_Clear := FALSE;
          SameSizeSlide_clear := FALSE; 
      END_IF
      
            Robot.M_StartMoveBoxToFeedInConveyor_ClampA(ConveyorSlideSelect := Info.ClampA_Setting.PlaceArea,
                                                        DiffSizeSlideClear  := DiffSizeSlide_Clear,
                                                        SameSizeSlideClear  := SameSizeSlide_clear);
        ELSE
      tonTimeOut.IN:=FALSE;
            uiExecutingStep := 99000; // Go to process end
        END_IF
    tonTimeOut.IN :=TRUE;   
    IF tonTimeOut.Q THEN
      tonTimeOut.IN:=FALSE;
      _Abort :=TRUE;    
      uiResumeStep:=61000;  
      strStatus :='Place Box timeout';
    END_IF
    70000: // Only ClampB place box
        // Clear command
        WareHouse.M_ResetReloadBox();
        Robot.M_ResetAllCommand();

        // Check robot RSR1 not working
        IF NOT Robot._DI1.Done AND NOT (Robot._DI1.AbsMoveA OR Robot._DI1.AbsMoveB OR Robot._DI1.WarehouseA OR Robot._DI1.WarehouseB) THEN
            uiExecutingStep := 71000;
        END_IF
    71000:
        IF NOT Robot._DI1.Done THEN
      IF NOT DiffSizeCV.InBackWard AND SameSizeCV.InBackWard THEN
        CASE Info.ClampA_Setting.PlaceArea OF
          E_FeedInEmptyBox_PlaceArea.DiffSizeConveyor:
          
                  DiffSizeCV.M_MoveForward();
          E_FeedInEmptyBox_PlaceArea.SameSizeConveyor:
            SameSizeCV.M_MoveForward();
        END_CASE

              IF input.bDifferentSizeCV_BoxDetect7_Sensor THEN
                  DiffSizeSlide_Clear := FALSE;
              ELSE
                  DiffSizeSlide_Clear := TRUE;
              END_IF

              IF Input.bSameSizeCV_BoxNearStorageSensor THEN
                  SameSizeSlide_clear := FALSE;
              ELSE
                  SameSizeSlide_clear := TRUE;
              END_IF
      ELSE
          DiffSizeSlide_Clear := FALSE;
          SameSizeSlide_clear := FALSE; 
      END_IF
            Robot.M_StartMoveBoxToFeedInConveyor_ClampB(ConveyorSlideSelect := Info.ClampB_Setting.PlaceArea,
                                                        DiffSizeSlideClear  := DiffSizeSlide_Clear,
                                                        SameSizeSlideClear  := SameSizeSlide_clear);
        ELSE
      tonTimeOut.IN:=FALSE;
            uiExecutingStep := 99000; // Go to process end
        END_IF
    tonTimeOut.IN :=TRUE;   
    IF tonTimeOut.Q THEN
      tonTimeOut.IN:=FALSE;
      _Abort :=TRUE;    
      uiResumeStep:=71000;  
      strStatus :='Place Box timeout';
    END_IF
    80000: // Both Clamp place box
        WareHouse.M_ResetReloadBox(); // Clear Warehouse reload command
        Robot.M_ResetAllCommand(); // Clear Fanuc Robot command
        IF NOT Robot._DI1.Done THEN
            uiExecutingStep := 81000;
        END_IF;
    81000:
      
        CASE uiPlaceBothStep OF
      
            0:                
                SlideClear_1st  := FALSE;
                SlideClear_2nd  := FALSE;
      IF NOT DiffSizeCV.InBackWard AND NOT SameSizeCV.InBackWard THEN
        CASE Info.ClampA_Setting.PlaceArea OF
          E_FeedInEmptyBox_PlaceArea.DiffSizeConveyor:
                  DiffSizeCV.M_MoveForward();
            uiPlaceBothStep := 10;
          E_FeedInEmptyBox_PlaceArea.SameSizeConveyor:
            SameSizeCV.M_MoveForward();
            uiPlaceBothStep := 10;
        END_CASE
      END_IF
            10:
                // ClampA place box
        
        CASE Info.ClampA_Setting.PlaceArea OF
          E_FeedInEmptyBox_PlaceArea.DiffSizeConveyor:
            IF NOT DiffSizeCV.InStopped  THEN
              DiffSizeCV.M_MoveForward();
            END_IF
            //uiPlaceBothStep := 10;
          E_FeedInEmptyBox_PlaceArea.SameSizeConveyor:
            IF  NOT SameSizeCV.InStopped  THEN
              SameSizeCV.M_MoveForward();
            END_IF
            //uiPlaceBothStep := 10;
        END_CASE

        
        IF  NOT DiffSizeCV.InStopped OR  NOT SameSizeCV.InStopped THEN
                  IF info.ClampA_Setting.PlaceArea = E_FeedInEmptyBox_PlaceArea.DiffSizeConveyor THEN
                      IF Input.bDifferentSizeCV_BoxDetect7_Sensor THEN
                          SlideClear_1st := FALSE;
                      ELSE
                          SlideClear_1st := TRUE;
                      END_IF

                  ELSIF info.ClampA_Setting.PlaceArea = E_FeedInEmptyBox_PlaceArea.SameSizeConveyor THEN
                      IF Input.bSameSizeCV_BoxNearStorageSensor THEN
                          SlideClear_1st := FALSE;
                      ELSE
                          SlideClear_1st := TRUE;
                      END_IF
                  END_IF
          IF SlideClear_1st AND NOT Robot._di1.ClampA_Sensor THEN
                    uiPlaceBothStep := 20;
          END_IF
        ELSE
          SlideClear_1st := FALSE;
        END_IF
            20:
        SlideClear_2nd := FALSE;
        tonPlaceSensorDelay.IN :=FALSE;
        IF NOT DiffSizeCV.InStopped THEN
          DiffSizeCV.M_MoveForward();
        END_IF
        IF NOT SameSizeCV.InStopped THEN
          SameSizeCV.M_MoveForward();
        END_IF
                IF ((info.ClampA_Setting.PlaceArea = E_FeedInEmptyBox_PlaceArea.DiffSizeConveyor) AND NOT Input.bDifferentSizeCV_BoxDetect7_Sensor) THEN
           uiPlaceBothStep := 30;
            //uiPlaceBothStep := 25;
                ELSIF ((info.ClampA_Setting.PlaceArea = E_FeedInEmptyBox_PlaceArea.SameSizeConveyor) AND NOT Input.bSameSizeCV_BoxDetect6_Sensor) THEN
                     uiPlaceBothStep := 30;
            //uiPlaceBothStep := 25;
                END_IF
        
        
            30:
						// ClampB place box
				CASE Info.ClampB_Setting.PlaceArea OF
				  E_FeedInEmptyBox_PlaceArea.DiffSizeConveyor:
					IF   DiffSizeCV.InStopped  THEN
					  DiffSizeCV.M_MoveForward();
					END_IF
					//uiPlaceBothStep := 10;
				  E_FeedInEmptyBox_PlaceArea.SameSizeConveyor:
					IF   SameSizeCV.InStopped  THEN
					  SameSizeCV.M_MoveForward();
					END_IF
					//uiPlaceBothStep := 10;
				END_CASE
				TON_DiffSizeCVmove.IN := DiffSizeCV.InForWard;		// make sure TransCV still moveforward; edit Gamin 20251117
				TON_SameSizeCVmove.IN := SameSizeCV.InForWard;
				IF NOT DiffSizeCV.InStopped OR NOT SameSizeCV.InStopped THEN
					   IF info.ClampB_Setting.PlaceArea = E_FeedInEmptyBox_PlaceArea.DiffSizeConveyor THEN
						 	IF Input.bDifferentSizeCV_BoxDetect7_Sensor THEN
							  	SlideClear_2nd := FALSE;
						   	ELSE                        
//              			tonPlaceSensorDelay.IN :=TRUE ;   //edit by min 20251028
								IF TON_DiffSizeCVmove.Q THEN
								  SlideClear_2nd := TRUE;
								END_IF
                       		END_IF
               			ELSIF info.ClampB_Setting.PlaceArea = E_FeedInEmptyBox_PlaceArea.SameSizeConveyor THEN
							 IF Input.bSameSizeCV_BoxNearStorageSensor THEN
								 SlideClear_2nd := FALSE;
							 ELSE
		//              tonPlaceSensorDelay.IN :=TRUE ; //edit by min 20251028
								IF TON_SameSizeCVmove.Q THEN
								  SlideClear_2nd := TRUE;
								END_IF
                     		END_IF
                   		END_IF
        		END_IF
        
        IF SlideClear_2nd THEN
                  uiPlaceBothStep := 99;
          tonPlaceSensorDelay.IN :=FALSE;
		  TON_DiffSizeCVmove.IN := FALSE;
		  TON_SameSizeCVmove.IN := FALSE;
        END_IF
      
            99:
        // wait reset
        END_CASE

        IF NOT Robot._DI1.Done THEN
            Robot.M_StartMoveBoxToFeedInConveyor_ClampBoth(ClampA_Address := info.ClampA_Setting.PlaceArea,
                                                           ClampB_Address := info.ClampB_Setting.PlaceArea,
                                                           SlideClear_1st := SlideClear_1st,
                                                           SlideClear_2nd := SlideClear_2nd);
        ELSE
      tonTimeOut.IN:=FALSE;
            uiExecutingStep := 99000;
        END_IF
    tonTimeOut.IN :=TRUE;   
    IF tonTimeOut.Q THEN
      tonTimeOut.IN:=FALSE;
      _Abort :=TRUE;  
      uiResumeStep:=81000;    
      strStatus :='Place Box timeout';
    END_IF
   99000: // process done
    // 持續檢測軌道是否在前進：
    // 每一個 PLC 掃描週期都會執行這一行
    // 若 InForWard = TRUE → TON 開始/持續計時
    // 若 InForWard = FALSE → TON 自動歸零(因為 IN=FALSE) → 下次再前進就重新計時
	SameSizeCV.M_MoveForward();
	DiffSizeCV.M_MoveForward();
    tonFeedInConveyorDelay.IN := DiffSizeCV.InForWard OR SameSizeCV.InForWard; // Delay FeedInConveyor stop 500ms

    //  當「連續前進時間」滿足 TON 設定的 PT，就會 Q=TRUE（同樣是每掃描都檢查）
    IF tonFeedInConveyorDelay.Q THEN
        // 時間到後要做的事：釋放權限 + 進下一步
        DAS_CoreSys.MachineControl.fballocatearea.M_ReleasePulloutAccess(
            ControlAccess := E_RoundBeltControlAccess.FanucRobot);

        //  現在改成：本 FB 不主動停馬達，讓別的地方決定要不要停
        // DiffSizeCV.M_MotorStop();
        // SameSizeCV.M_MotorStop();

        tonFeedInConveyorDelay.IN := FALSE; // 用完這次計時就清掉，等下次需要再開
        Status          := 'Wait box move leave sensor ';
        uiExecutingStep := 99100;
    END_IF

  99100:
      Status    := 'Process completed';
      DiffSizeCV.M_MotorStop();
      SameSizeCV.M_MotorStop();
      IF DiffSizeCV.InStopped AND SameSizeCV.InStopped THEN
         _Executed := TRUE;
      END_IF
END_CASE

IF _Executed THEN
    eState := STATE_DONE;
ELSIF NOT Execute THEN
    eState := STATE_RESETTING;
ELSIF Abort OR _Abort THEN
  //FUN_UniqueErrorCodeGenerator(iErrorID := ErrorID,UinqueErrorCode=>_UniqueErrorCode);
  eState := STATE_ABORTING;
ELSIF _Error THEN
  //FUN_UniqueErrorCodeGenerator(iErrorID := ErrorID,UinqueErrorCode=>_UniqueErrorCode);
  eState := STATE_ERROR;
  
END_IF
END_METHOD

METHOD  M_STATE_RESETTING
VAR_INPUT
END_VAR
IF _Executed THEN Done :=TRUE ; END_IF
CASE uiResettingStep OF
	0:
		TON_DiffSizeCVmove.IN := FALSE;
		TON_SameSizeCVmove.IN := FALSE;
		//DAS.fbStorageArea.M_InactivePulloutConveyorInternCtrl();
		Robot.M_ResetAllCommand();
		Robot.Bzone_AllowWork:=FALSE;
		DiffSizeCV.M_MotorStop();
		SameSizeCV.M_MotorStop();
		 DAS_CoreSys.MachineControl.fballocatearea.M_ReleasePulloutAccess(ControlAccess := E_RoundBeltControlAccess.FanucRobot);
		 DAS_CoreSys.MachineControl.fballocatearea.M_StopStoragePulloutAction();
		WareHouse.M_ResetFeedInBox();
		WareHouse.M_ResetReloadBox();
		uiResettingStep := 100;
	100:
		_ResetCompleted := TRUE;
END_CASE
IF _ResetCompleted THEN
    eState := STATE_DORMANT;
END_IF
END_METHOD

END_FUNCTION_BLOCK

// ---- Library/20_MachineUnits/21_StorageArea/Old_version_Service/FB_FeedInRoundBeltBoxBatch_Old.TcPOU
// ═══════════════════════════════════════════════════════════════════════════
// FB_FeedInRoundBeltBoxBatch
// 圓帶回倉 — 批次服務 FB
// ═══════════════════════════════════════════════════════════════════════════
//
// 【用途】
// 管理最多 40 筆「從圓帶取盒回倉儲 / 或放到 PullOut」流程,每筆由
// FB_FeedInRoundBeltBoxToWareHouse (HandshakeMode=TRUE) 逐筆執行。
// 每筆 flow 可獨立決定目的地: WareHouseA / WareHouseB / PullOutInner / PullOutOuter
//
// 【設計模式】
// 仿 FB_WareHouseInnerPickToRoundBeltBatch:
//   1. 收到 Execute → 迭代 FlowInfo[0..NrOfFlow-1]
//   2. 跳過無效項 (ID = -1 或 A/B 爪皆 NoWork)
//   3. 對每筆有效流程配置並啟動 fbSingleFlow,等其完成/失敗
//   4. 每筆完成後 PLC 透過 FeedBack/ReadComplete 等 C# 讀完 ActionRecords 才進下一筆
//   5. 跨迭代強制清 handshake 防 C# 遺漏
//
// 【FeedBack / ReadComplete 握手協定】
// 同 FB_WareHouseInnerPickToRoundBeltBatch:
//   PLC: 單筆完成 → FeedBack:=TRUE → 等 ReadComplete=TRUE → 清 FeedBack → 進下一筆
//   C#:  看到 FeedBack=TRUE → 讀 ActionRecords → 寫 ReadComplete=TRUE → 等 FeedBack=FALSE → 清 ReadComplete
//
// 【Resume / Pause】
// Resume: 錯誤後 C# 按 Reset → 從 uiResumeStep 繼續 (固定回 100 重新配置 fbSingleFlow)
// Pause:  僅在迭代邊界 (step 0 / 310) 生效, 不中斷單筆流程
//
// Create Date : 2026/04/14
// ═══════════════════════════════════════════════════════════════════════════

FUNCTION_BLOCK FB_FeedInRoundBeltBoxBatch_Old EXTENDS FB_ObjectBase_V2 IMPLEMENTS IBasicElement

VAR_INPUT
	// ----- 外部資源參照 -----
	Robot			: REFERENCE TO FB_FanucRobot_Basic_V2;	// 倉儲區 Fanuc 手臂
	RoundBelt		: REFERENCE TO FB_RoundBeltService;		// 圓帶服務
	WareHouse		: REFERENCE TO FB_WareHouse;				// 倉儲 FB
	Input			: ST_InputTable;						// IO 輸入表

	// ----- 批次資料 (C# HMI ↔ PLC 介面) -----
	BatchInfo		: REFERENCE TO ST_FeedInRBBatch;

	Stop			: BOOL;									// 外部停止信號
END_VAR

VAR_OUTPUT
END_VAR

VAR
	// ----- 狀態與錯誤追蹤 -----
	strStatus			: STRING;
	tonTimeOut			: TON;				// Per-iteration 逾時 (PT=600s, step 310 推進時重置)
	_UniqueErrorCode	: STRING;
	uiResumeStep		: UDINT := 0;
	_bRetry				: BOOL;

	// ----- 批次迭代控制 -----
	iProcessingIndex	: INT := 0;
	CurrentFlow			: ST_FeedInRBFlowInfo;

	// ----- 內嵌單筆 FB -----
	fbSingleFlow		: FB_FeedInRoundBeltBoxToWareHouse;
	_bSingleFlowStarted	: BOOL;
END_VAR

// ============================================================
// 執行順序: input piping → A00 → A10 → output piping
// ============================================================

// 1. Input piping: C# → fbSingleFlow
IF __ISVALIDREF(BatchInfo) THEN
	fbSingleFlow.ReadComplete := BatchInfo.ReadComplete;
	Execute := BatchInfo.HandShake.Execute;
	Reset	:= BatchInfo.HandShake.Reset;
END_IF

// 2. Timer PT setup
A00_BasicUnits();

// 3. State machine
SUPER^.A10_StateControl();

// 4. Output piping: fbSingleFlow → C#
IF __ISVALIDREF(BatchInfo) THEN
	BatchInfo.ActionRecords := fbSingleFlow.ActionRecords;
	BatchInfo.ActionIndex := fbSingleFlow.ActionIndex;
	BatchInfo.FeedBack := fbSingleFlow.FeedBack;
	BatchInfo.HandShake.Done := Done;
	BatchInfo.HandShake.Busy := Busy;
	BatchInfo.HandShake.Error := Error;
END_IF

ACTION A00_BasicUnits:
// Per-iteration timeout, step 310 推進時重置
tonTimeOut(PT := T#600S);

fbSingleFlow(Input := Input);
END_ACTION

// 尋找下一筆有效流程
// 從 iProcessingIndex 開始往後掃描 BatchInfo.FlowInfo[]
// 有效條件: ID <> -1 且至少一爪為 Work
// 無效流程自動跳過並記錄 WorkedID
// 回傳 TRUE = 找到有效流程 (iProcessingIndex 已更新), FALSE = 全部完成
METHOD M_FindNextValidFlow : BOOL
VAR_INPUT
END_VAR
VAR
	i		: INT;
	bValid	: BOOL;
END_VAR
IF NOT __ISVALIDREF(BatchInfo) THEN
	M_FindNextValidFlow := FALSE;
	RETURN;
END_IF

IF BatchInfo.NrOfFlow = 0 THEN
	M_FindNextValidFlow := FALSE;
	RETURN;
END_IF

FOR i := iProcessingIndex TO UINT_TO_INT(BatchInfo.NrOfFlow) - 1 BY 1 DO
	bValid := FALSE;

	IF BatchInfo.FlowInfo[i].ID <> -1 THEN
		IF BatchInfo.FlowInfo[i].ClampA_Setting.Behavior = E_ClampWork.Work
		OR BatchInfo.FlowInfo[i].ClampB_Setting.Behavior = E_ClampWork.Work THEN
			bValid := TRUE;
		END_IF
	END_IF

	IF bValid THEN
		iProcessingIndex := i;
		CurrentFlow := BatchInfo.FlowInfo[i];
		M_FindNextValidFlow := TRUE;
		RETURN;
	ELSE
		BatchInfo.WorkedID[i] := BatchInfo.FlowInfo[i].ID;
	END_IF
END_FOR

M_FindNextValidFlow := FALSE;
END_METHOD

// 已中止狀態 — 等待 Reset 信號
METHOD M_STATE_ABORTED
VAR_INPUT
END_VAR
IF NOT _bRetry THEN
	Busy 	:= FALSE;
	Aborted := TRUE;
	Error 	:= TRUE;
	Status 	:= strStatus;
	uiAbortingStep := 0;
	_AbortCompleted := FALSE;
END_IF
// 判斷內部Serivce 已經在aborted 狀態等著才能讓 FB reset
IF fbSingleFlow.eState = STATE_Aborted THEN
	IF reset THEN
		fbSingleFlow();
		fbSingleFlow.Reset := TRUE;

		_bRetry := TRUE;
		Aborted	:= FALSE;
		Error	:= FALSE;
	END_IF
END_IF

// 狀態機切換
IF NOT Execute THEN
	eState := STATE_RESETTING;
ELSIF Execute AND _bRetry THEN
	IF fbSingleFlow.eState = STATE_EXECUTING OR fbSingleFlow.eState = STATE_DONE THEN
		fbSingleFlow.Reset := FALSE;
		IF uiResumeStep > 0 THEN
			status			:= '';
			uiExecutingStep := uiResumeStep;
			eState 			:= STATE_EXECUTING;
		END_IF
	END_IF
END_IF


//IF __ISVALIDREF(BatchInfo) THEN
//	IF BatchInfo.HandShake.Reset THEN
//		IF uiResumeStep > 0 THEN
//			uiExecutingStep := uiResumeStep;
//			_bRetry := TRUE;
//		END_IF
//		eState := STATE_RESETTING;
//	END_IF
//ELSIF Reset THEN
//	IF uiResumeStep > 0 THEN
//		uiExecutingStep := uiResumeStep;
//		_bRetry := TRUE;
//	END_IF
//	eState := STATE_RESETTING;
//END_IF
END_METHOD

// 中止狀態 — 先停止單筆 FB
METHOD M_STATE_ABORTING
VAR_INPUT
END_VAR
CASE uiAbortingStep OF
	0:
		_Abort := FALSE;
		_bRetry := FALSE;
		tonTimeOut.IN := FALSE;
		IF _bSingleFlowStarted THEN
			fbSingleFlow.Abort := TRUE;
			fbSingleFlow();
		END_IF
		uiAbortingStep := 100;
	
	100:
		fbSingleFlow();
		IF fbSingleFlow.Aborted OR NOT fbSingleFlow.Busy THEN
			fbSingleFlow.Abort := FALSE;
			uiAbortingStep := 9999;
		END_IF
	
	9999:
		_AbortCompleted := TRUE;
END_CASE

IF NOT Execute THEN
	eState := STATE_RESETTING;
ELSIF Execute AND _AbortCompleted THEN
	eState := STATE_Aborted;
END_IF
END_METHOD

// 完成狀態 — 等待外部取消 Execute
METHOD M_STATE_DONE
VAR_INPUT
END_VAR
Busy := FALSE;
Done := TRUE;

IF __ISVALIDREF(BatchInfo) THEN
	IF NOT BatchInfo.HandShake.Execute THEN
		eState := STATE_RESETTING;
	END_IF
ELSIF NOT Execute THEN
	eState := STATE_RESETTING;
END_IF
END_METHOD

// 休眠狀態 — 清除旗標,監聽 BatchInfo.HandShake.Execute 觸發
METHOD M_STATE_DORMANT
VAR_INPUT
END_VAR
Busy				:= FALSE;
Done				:= FALSE;
Aborted				:= FALSE;
Error				:= FALSE;
ErrorID				:= 0;
Status				:= '';
_ResetCompleted		:= FALSE;
_Error				:= FALSE;
_Executed			:= FALSE;
_Abort				:= FALSE;
uiExecutingStep		:= 0;
uiResettingStep		:= 0;
uiResumeStep		:= 0;
uiAbortingStep		:= 0;

tonTimeOut.IN		:= FALSE;
_UniqueErrorCode	:= '0';

iProcessingIndex	:= 0;
_bSingleFlowStarted	:= FALSE;

IF __ISVALIDREF(BatchInfo) THEN
	MEMSET(ADR(BatchInfo.WorkedID), 0, SIZEOF(BatchInfo.WorkedID));
END_IF

_AbortCompleted		:= FALSE;
_bRetry				:= FALSE;

IF Execute THEN
	eState := STATE_EXECUTING;
END_IF

//IF __ISVALIDREF(BatchInfo) THEN
//	IF BatchInfo.HandShake.Execute AND NOT Stop THEN
//		Execute := TRUE;
//		eState := STATE_EXECUTING;
//	END_IF
//	IF BatchInfo.HandShake.Reset THEN
//		Reset := TRUE;
//	END_IF
//END_IF
END_METHOD

// 錯誤狀態 — 顯示錯誤訊息
METHOD M_STATE_ERROR
VAR_INPUT
END_VAR
Busy := FALSE;
Error := TRUE;
Status := strStatus;

IF NOT Execute THEN
	eState := STATE_RESETTING;
END_IF

//IF __ISVALIDREF(BatchInfo) THEN
//	IF NOT BatchInfo.HandShake.Execute THEN
//		eState := STATE_RESETTING;
//	END_IF
//ELSIF NOT Execute THEN
//	eState := STATE_RESETTING;
//END_IF
END_METHOD

// 執行主狀態 — 迭代批次中每筆有效流程
// 步序:
//   0:      M_FindNextValidFlow → 找到跳 100 / 沒找到跳 99000
//   100:    強制清 handshake + 配置 fbSingleFlow + 啟動 (HandshakeMode := TRUE)
//   200:    每 cycle 呼叫 fbSingleFlow, 等 Done 跳 300, 等 Error/Aborted abort
//   300:    寫 WorkedID + 強制清 ReadComplete + 釋放 fbSingleFlow
//   310:    等 fbSingleFlow 回 DORMANT, iProcessingIndex+1, 重置 timer 回 0
//   99000:  全部完成
METHOD M_STATE_EXECUTING
VAR_INPUT
END_VAR
Busy := TRUE;
tonTimeOut.IN := TRUE;

// 非自動模式直接中止
IF GVL_Machine.PackTags[UnitNo.Storage].Status.UnitModeCurrent <> E_UnitMode.Auto THEN
	strStatus := 'Not in Auto mode';
	_UniqueErrorCode := 'E_NOT_AUTO_MODE';
	_Abort := TRUE;
END_IF

// Pause: 僅在迭代邊界 (step 0/310) 生效
IF __ISVALIDREF(BatchInfo) AND BatchInfo.Pause THEN
	IF uiExecutingStep = 0 OR uiExecutingStep = 310 THEN
		strStatus := 'Paused (at iteration boundary)';
	END_IF
END_IF

// Per-iteration timeout (600s, step 310 推進時重置)
IF tonTimeOut.Q THEN
	strStatus := 'Batch per-iteration timeout';
	_UniqueErrorCode := 'E_BATCH_TIMEOUT';
	uiResumeStep := 100;
	_Abort := TRUE;
END_IF

CASE uiExecutingStep OF

// ===== Step 0: 尋找下一筆有效流程 =====
0:
	IF NOT M_FindNextValidFlow() THEN
		uiExecutingStep := 99000;
	ELSE
		strStatus := CONCAT('Processing flow #', INT_TO_STRING(iProcessingIndex));
		uiExecutingStep := 100;
	END_IF

// ===== Step 100: 配置並啟動單筆 FB =====
100:
	// Safety: 強制清 handshake 確保 C# 看到本迭代 FeedBack 上升緣
	IF __ISVALIDREF(BatchInfo) THEN
		BatchInfo.FeedBack := FALSE;
		BatchInfo.ReadComplete := FALSE;
	END_IF
	fbSingleFlow.ReadComplete := FALSE;

	// 配置參照與 input
	fbSingleFlow.Robot REF= Robot;
	fbSingleFlow.RoundBelt REF= RoundBelt;
	fbSingleFlow.WareHouse REF= WareHouse;
	fbSingleFlow.Input := Input;
	fbSingleFlow.Info.ClampA_Setting := CurrentFlow.ClampA_Setting;
	fbSingleFlow.Info.ClampB_Setting := CurrentFlow.ClampB_Setting;
	fbSingleFlow.Stop := Stop;
	fbSingleFlow.HandshakeMode := TRUE;	// 啟用 ActionRecord + FeedBack/ReadComplete
	fbSingleFlow.Execute := TRUE;
	_bSingleFlowStarted := TRUE;
	uiExecutingStep := 200;

// ===== Step 200: 等待單筆 FB 完成 =====
200:
	fbSingleFlow();
	IF fbSingleFlow.Done THEN
		uiExecutingStep := 300;
	ELSIF fbSingleFlow.Error OR fbSingleFlow.Aborted THEN
		strStatus := CONCAT('Flow #', CONCAT(INT_TO_STRING(iProcessingIndex), ' failed'));
		_UniqueErrorCode := 'E_FLOW_FAILED';
		uiResumeStep := 100;	// retry 從重配置開始
		_Abort := TRUE;
	END_IF

// ===== Step 300: 記錄完成 + 釋放單筆 FB =====
300:
	IF __ISVALIDREF(BatchInfo) THEN
		BatchInfo.WorkedID[iProcessingIndex] := CurrentFlow.ID;
		BatchInfo.ReadComplete := FALSE;	// Safety: 防 C# 殘留
	END_IF
	fbSingleFlow.Execute := FALSE;
	fbSingleFlow();
	_bSingleFlowStarted := FALSE;
	uiExecutingStep := 310;

// ===== Step 310: 等 fbSingleFlow 回 DORMANT 後再推進 =====
310:
	fbSingleFlow();
	IF NOT fbSingleFlow.Busy AND NOT fbSingleFlow.Done AND NOT fbSingleFlow.Error THEN
		iProcessingIndex := iProcessingIndex + 1;
		tonTimeOut.IN := FALSE;	// per-iteration timer 重置
		uiExecutingStep := 0;
	END_IF

// ===== Step 99000: 全部完成 =====
99000:
	_Executed := TRUE;

END_CASE

// ===== 狀態切換 =====
IF NOT Execute THEN
	eState := STATE_RESETTING;
ELSIF _Error THEN
	eState := STATE_ERROR;
ELSIF _Abort THEN
	eState := STATE_ABORTING;
ELSIF _Executed THEN
	eState := STATE_DONE;
END_IF
END_METHOD

// 重置狀態 — 等待 fbSingleFlow 回 DORMANT 後決定走 retry 或正常路徑
METHOD M_STATE_RESETTING
VAR_INPUT
END_VAR
CASE uiResettingStep OF
	0:
		//Done := FALSE;	//done 留到dormant 關閉。
		Error := FALSE;
		Aborted := FALSE;
		tonTimeOut.IN := FALSE;
	
		fbSingleFlow();
		fbSingleFlow.Execute := FALSE;
		uiResettingStep := 50;
	
	50:
		// 等 fbSingleFlow 真的回 DORMANT, 避免 race
//		fbSingleFlow.Reset := FALSE;
//		fbSingleFlow();
//		IF NOT fbSingleFlow.Busy AND NOT fbSingleFlow.Done AND NOT fbSingleFlow.Error AND NOT fbSingleFlow.Aborted THEN
//			IF _bRetry THEN
//				_bRetry := FALSE;
//				eState := STATE_EXECUTING;
//				RETURN;
//			END_IF
//			uiResettingStep := 100;
//		END_IF
		IF fbSingleFlow.eState = STATE_DORMANT THEN
			uiResettingStep := 100;
		END_IF
	
	100:
		_ResetCompleted := TRUE;
	
END_CASE

IF _ResetCompleted THEN
	eState := STATE_DORMANT;
END_IF
END_METHOD

END_FUNCTION_BLOCK

// ---- Library/20_MachineUnits/21_StorageArea/Old_version_Service/FB_FeedInRoundBeltBoxToWareHouse_Old.TcPOU
(*
	FB_FeedInRoundBeltBoxToWareHouse
	功能：從圓帶取盒子放回倉儲 (與 FB_ReloadRoundBeltBoxWithRobot_V2 反向操作)
	流程：圓帶移動到站位 → 手臂 AbsMove 從圓帶取盒 → 手臂放盒到倉儲
	安全卡控：手臂進入圓帶區域時，取得圓帶控制權，圓帶不可移動
*)
FUNCTION_BLOCK FB_FeedInRoundBeltBoxToWareHouse_Old EXTENDS FB_ObjectBase_V2 IMPLEMENTS IBasicElement
VAR_INPUT
    // ===== 外部元件參考 =====
    Robot         : REFERENCE TO FB_FanucRobot_Basic_V2; // Fanuc 手臂
	RoundBelt	  : REFERENCE TO FB_RoundBeltService;    // 圓帶服務
    WareHouse     : REFERENCE TO FB_WareHouse;           // 倉儲區
	Input         : ST_InputTable;                        // IO 輸入表
    Info          : ST_FeedInToWareHouseBox_Info;         // C# ADS 餵入的動作參數 (A爪/B爪 取盒位置、放盒目標)
    Stop          : BOOL;                                 // 停止訊號，暫停 Timeout 計時
//	Pause		  : BOOL;
END_VAR
VAR_OUTPUT
//	Paused		  : BOOL;
	AClampMoveDone	: BOOL;  // A爪動作完成旗標，供 C# 寫入 SQL
	BClampMoveDone	: BOOL;  // B爪動作完成旗標，供 C# 寫入 SQL
END_VAR
VAR
//	_Abort			  : BOOL;
    strStatus         : STRING;   // 錯誤/狀態訊息
    tonTimeOut        : TON;      // 通用逾時計時器 (120s)
    _UniqueErrorCode  : STRING;
    PreviousStrStatus : STRING;   // Resume 前的狀態訊息
    PreviousErrorCode : STRING;   // Resume 前的錯誤碼
    A2_Sensor         : BOOL;    // 圓帶 A2 位置感測器
    A3_Sensor         : BOOL;    // 圓帶 A3 位置感測器

	// ===== 爪工作旗標 =====
	_AClampDoingWork	: BOOL;  // A爪正在執行
	_BClampDoingWork	: BOOL;  // B爪正在執行

	// ========== Resume 續做機制 ==========
	uiResumeStep	: UDINT := 0;	// 錯誤發生時記錄的步驟，供續做使用
	
	// =========== Aborted =================
	_bRetry			: BOOL;
	
END_VAR

SUPER^.A10_StateControl();
A00_BasicUnits();
A2_Sensor := Input.bRoundBelt_ChangeZoneA2Detect_Sensor;
A3_Sensor := Input.bRoundBelt_ChangeZoneA3Detect_Sensor;

(*============================================================
Create Date : 2026/03/18
Last Update	: 2026/03/23
Change Log  : 2026/03/18，Initial version - Pick box from RoundBelt and place to WareHouse
			  2026/03/23，修正續做，新增手臂先在aborting清除錯誤，
			  2026/04/14，新的FB新增回拔輸送帶放盒位置支援，ActionRecords功能，把這一隻舊的移除。
============================================================*)

ACTION A00_BasicUnits:
tonTimeOut(PT:=T#120S);
END_ACTION

METHOD M_CheckCommand : BOOL
VAR_INPUT
END_VAR
VAR_INST
	CheckBehavior : BOOL;
END_VAR
VAR
	I: INT;
END_VAR
// Memory clear
CheckBehavior := FALSE;
// Check command is correct
IF info.ClampA_Setting.Behavior = E_ClampWork.Work OR info.ClampB_Setting.Behavior = E_ClampWork.Work THEN
	CheckBehavior := TRUE;
ELSE
	CheckBehavior := FALSE;
END_IF

M_CheckCommand := CheckBehavior;
END_METHOD

METHOD M_CheckUnitsNotBusy : BOOL
VAR_INPUT
END_VAR
M_CheckUnitsNotBusy := true;
END_METHOD

METHOD M_CheckUnitsReady : BOOL
VAR_INPUT
END_VAR
M_CheckUnitsReady := true;
END_METHOD

(* 根據 A爪/B爪 的 Behavior 和 PlaceArea 判斷動作模式
   - 單爪A/B：從圓帶取盒後放到 WareHouseA 或 WareHouseB
   - 雙爪：兩爪各自從圓帶取盒，放到指定的倉儲 (可同倉或不同倉)
*)
METHOD M_SelectActionMode : E_FeedInToWareHouseAction
VAR_INPUT
END_VAR
// 判斷 A爪/B爪 是否有工作，以及放盒目標倉儲
IF info.ClampA_Setting.Behavior <> E_ClampWork.Work AND info.ClampB_Setting.Behavior <> E_ClampWork.Work THEN
	M_SelectActionMode := E_FeedInToWareHouseAction.Undefined;
ELSIF info.ClampA_Setting.Behavior = E_ClampWork.Work AND info.ClampB_Setting.Behavior <> E_ClampWork.Work THEN
	IF info.ClampA_Setting.PlaceArea = E_FeedInToWareHouse_PlaceArea.WareHouseA THEN
		M_SelectActionMode := E_FeedInToWareHouseAction.ClampA_WareHouseA;
	ELSIF info.ClampA_Setting.PlaceArea = E_FeedInToWareHouse_PlaceArea.WareHouseB THEN
		M_SelectActionMode := E_FeedInToWareHouseAction.ClampA_WareHouseB;
	END_IF
ELSIF info.ClampA_Setting.Behavior <> E_ClampWork.Work AND info.ClampB_Setting.Behavior = E_ClampWork.Work THEN
	IF info.ClampB_Setting.PlaceArea = E_FeedInToWareHouse_PlaceArea.WareHouseA THEN
		M_SelectActionMode := E_FeedInToWareHouseAction.ClampB_WareHouseA;
	ELSIF info.ClampB_Setting.PlaceArea = E_FeedInToWareHouse_PlaceArea.WareHouseB THEN
		M_SelectActionMode := E_FeedInToWareHouseAction.ClampB_WareHouseB;
	END_IF
ELSIF info.ClampA_Setting.Behavior = E_ClampWork.Work AND info.ClampB_Setting.Behavior = E_ClampWork.Work THEN
	IF info.ClampA_Setting.PlaceArea = E_FeedInToWareHouse_PlaceArea.WareHouseA THEN
		IF info.ClampB_Setting.PlaceArea = E_FeedInToWareHouse_PlaceArea.WareHouseA THEN
			M_SelectActionMode := E_FeedInToWareHouseAction.A_WareHouseA_B_WareHouseA;
		ELSIF info.ClampB_Setting.PlaceArea = E_FeedInToWareHouse_PlaceArea.WareHouseB THEN
			M_SelectActionMode := E_FeedInToWareHouseAction.A_WareHouseA_B_WareHouseB;
		END_IF
	ELSIF info.ClampA_Setting.PlaceArea = E_FeedInToWareHouse_PlaceArea.WareHouseB THEN
		IF info.ClampB_Setting.PlaceArea = E_FeedInToWareHouse_PlaceArea.WareHouseA THEN
			M_SelectActionMode := E_FeedInToWareHouseAction.A_WareHouseB_B_WareHouseA;
		ELSIF info.ClampB_Setting.PlaceArea = E_FeedInToWareHouse_PlaceArea.WareHouseB THEN
			M_SelectActionMode := E_FeedInToWareHouseAction.A_WareHouseB_B_WareHouseB;
		END_IF
	END_IF
END_IF
END_METHOD

METHOD  M_STATE_ABORTED
VAR_INPUT
END_VAR
IF NOT _bRetry THEN
	Busy    := FALSE;
	Error	:= TRUE;
	Aborted := TRUE;
	UniqueErrorCode := _UniqueErrorCode;
	uiAbortingStep  := 0;
	_AbortCompleted := FALSE;
	Status := strStatus;
END_IF

IF reset THEN
	_bRetry := TRUE;
	Error	:= FALSE;
	Aborted := FALSE;
	_Abort  := FALSE;
END_IF

// ============================================================
// Resume 續做機制：保持 Execute 並按 Reset 可從錯誤點繼續執行
// ============================================================
IF NOT Execute THEN
	eState := STATE_RESETTING;
ELSIF Execute AND _bRetry AND NOT Robot._DI1.Error AND NOT Robot.Halt THEN
	// Resume 模式：確認 Robot 不在暫停且無錯誤，從儲存的步驟繼續執行
	Status := '';
	uiExecutingStep := uiResumeStep;
	PreviousStrStatus := strStatus;
	PreviousErrorCode := _UniqueErrorCode;
	IF GVL_ADS.MachineState <>E_MachineState.Error THEN
		eSTATE:=STATE_EXECUTING;
	END_IF
END_IF
END_METHOD

METHOD  M_STATE_ABORTING
VAR_INPUT
END_VAR
CASE uiAbortingStep OF 
	0:
			_Abort 				:= FALSE;
			_bRetry				:= FALSE;
			tonTimeOut.IN 		:= FALSE;

			// 清除 Robot DO handshake 和周邊狀態（不管 Robot 是 Error 還是 Held）
	
			(* 
				comment edited By Gamin ，
				1. 續做不能清除手臂命令，如果是做雙爪夾盒，A爪做完B爪報錯進入到續做流程，如果在此清除掉手臂命令
					，後續回到executing 動作，此時的情境為A 已做完已夾完盒，等同於給手臂重新做的命令，，會有危險，
				2. 在Service 執行期間進入到錯誤狀態也不能清除圓帶的使用權，以免被其他的Serivce 搶走，會有危險
				3.  A、B done 不能清除，這旗標也可算是代表手臂該爪的動作完成，
				   如果A爪完成，B爪報錯，續做只接續著做B爪，這樣Service 結束就只會有B done。
			*)
//			Robot.M_ResetAllCommand();
//			WareHouse.M_ResetFeedInBox();
//			DAS_CoreSys.MachineControl.fbAllocateArea.M_ResetReloadRoundBeltAction();
//			DAS_CoreSys.MachineControl.fbAllocateArea.M_ReleaseRoundBeltAccess(ControlAccess := E_RoundBeltControlAccess.FanucRobot);
//			AClampMoveDone	 := FALSE;
//			BClampMoveDone	 := FALSE;
//			_AClampDoingWork := FALSE;
//			_BClampDoingWork := FALSE;

			uiAbortingStep := 100;
    100:
			IF Robot._DI1.Error THEN
				uiAbortingStep := 200;
			ELSE
				uiAbortingStep := 9999;
			END_IF
			
	200:		
			 IF DAS_CoreSys.MachineControl.M_RobotResetCmd() THEN
				 uiAbortingStep := 300;
			 END_IF
			 
	300:
			IF DAS_CoreSys.MachineControl.M_RobotStartCmd() THEN
				 uiAbortingStep := 400;
			 END_IF 
			 
	400:
			IF Robot._DI1.Error THEN
		 		uiAbortingStep := 200;
			ELSE
				uiAbortingStep := 9999;
			END_IF
			
	9999:
			_AbortCompleted := TRUE;
END_CASE


IF _AbortCompleted THEN
    eState := STATE_Aborted;
END_IF
END_METHOD

METHOD  M_STATE_DONE
VAR_INPUT
END_VAR
Busy := FALSE;
Done := TRUE;
IF NOT Execute THEN
    eState := STATE_RESETTING;
END_IF
END_METHOD

METHOD  M_STATE_DORMANT
VAR_INPUT
END_VAR
// 清除 FB 所有輸出與內部狀態
Busy            := FALSE;
Done            := FALSE;
Aborted         := FALSE;
Error           := FALSE;
ErrorID         := 0;
Status          := '';
_ResetCompleted := FALSE;
_Error          := FALSE;
_Executed       := FALSE;
_Abort			:= FALSE;

uiExecutingStep := 0;
uiAbortingStep	:= 0;
uiResettingStep := 0;
uiResumeStep    := 0;

tonTimeOut.IN := FALSE;

PreviousStrStatus := '';
PreviousErrorCode := '';
_UniqueErrorCode := '0';

AClampMoveDone 	 := FALSE;
BClampMoveDone 	 := FALSE;
_AClampDoingWork := FALSE;
_BClampDoingWork := FALSE;
_AbortCompleted	 := FALSE;

_bRetry			:= FALSE;

// 等待 Execute 命令啟動
IF Execute AND NOT Stop THEN
    eState := STATE_EXECUTING;
END_IF
END_METHOD

METHOD  M_STATE_ERROR
VAR_INPUT
END_VAR
UniqueErrorCode	:= _UniqueErrorCode;
Error			:= TRUE;
status			:= strStatus;
Busy			:= FALSE;

IF NOT Execute THEN
    eState := STATE_RESETTING;
END_IF
END_METHOD

(*
	M_STATE_EXECUTING 主執行流程
	Step 配置：
	  0~1100    : 初始化、命令檢查、模式選擇
	  10000~10080 : A爪單爪 - 從圓帶取盒
	  20000~20080 : B爪單爪 - 從圓帶取盒
	  30000~31080 : 雙爪 - 從圓帶取盒 (先A後B，支援同站/不同站)
	  60000~61080 : A爪單爪 - 放盒到倉儲
	  70000~71080 : B爪單爪 - 放盒到倉儲
	  80000~81000 : 雙爪 - 放盒到倉儲 (支援同倉/不同倉)
	  99000       : 流程完成
*)
METHOD M_STATE_EXECUTING
VAR_INPUT
END_VAR
VAR_INST
    ActionMode       : E_FeedInToWareHouseAction;   // 動作模式 (單爪A/B、雙爪 × 目標倉儲)
	BoxReady_1st     : BOOL;  // 第一個盒子就緒 (A爪用)
	BoxReady_2nd     : BOOL;  // 第二個盒子就緒 (B爪用)
    CarrierReady_1st : BOOL;  // 第一個載具就緒
    CarrierReady_2nd : BOOL;  // 第二個載具就緒
    uiPickUpBothStep : UINT;  // 雙爪取盒子步驟
    uiPlaceBothStep  : UINT;  // 雙爪放盒子步驟
    ClampA_WareHouseCoordinates : ST_WareHouseCoordinates;  // A爪倉儲目標座標 (Layer/Slide)
    ClampB_WareHouseCoordinates : ST_WareHouseCoordinates;  // B爪倉儲目標座標 (Layer/Slide)
END_VAR
// Set status busy
Busy := TRUE;
IF THIS^.Stop THEN // Pending the timeout when Stop signal occur
	tonTimeout.IN :=FALSE;
END_IF
CASE uiExecutingStep OF
    0: // 初始化變數
        ActionMode       := E_FeedInToWareHouseAction.Undefined;
        CarrierReady_1st := FALSE;
        CarrierReady_2nd := FALSE;
        uiPickUpBothStep := 0;
        uiPlaceBothStep  := 0;
		BoxReady_1st := FALSE;
		BoxReady_2nd := FALSE;
        // 確認命令是否正確 (至少一個爪有 Work)
        IF M_CheckCommand() THEN
            uiExecutingStep := 10;
		ELSE
			strStatus := 'FB_FeedInRoundBeltBoxToWareHouse ,Step 0 : CheckCommand Error';
			_Error := TRUE;
        END_IF
    10: // 確認各元件就緒
        IF M_CheckUnitsReady() THEN
            uiExecutingStep := 20;
        END_IF
    20: // 確認各元件未忙碌
        IF M_CheckUnitsNotBusy() THEN
            uiExecutingStep := 1000;
        END_IF
    1000: // 根據 Info 選擇動作模式
        ActionMode      := M_SelectActionMode();
        uiExecutingStep := 1100;
    1100: // 取得圓帶控制權 (安全卡控：手臂進入圓帶區域，圓帶不可移動)
		DAS_CoreSys.MachineControl.fbAllocateArea.M_GetRoundBeltAccess(ControlAccess := E_RoundBeltControlAccess.FanucRobot);
		// 依動作模式跳轉對應步驟
        CASE ActionMode OF
            E_FeedInToWareHouseAction.ClampA_WareHouseA,
            E_FeedInToWareHouseAction.ClampA_WareHouseB:
                uiExecutingStep := 10000;  // A爪單爪取盒
            E_FeedInToWareHouseAction.ClampB_WareHouseA,
            E_FeedInToWareHouseAction.ClampB_WareHouseB:
                uiExecutingStep := 20000;  // B爪單爪取盒
            E_FeedInToWareHouseAction.A_WareHouseA_B_WareHouseA,
            E_FeedInToWareHouseAction.A_WareHouseA_B_WareHouseB,
            E_FeedInToWareHouseAction.A_WareHouseB_B_WareHouseA,
            E_FeedInToWareHouseAction.A_WareHouseB_B_WareHouseB:
                uiExecutingStep := 30000;  // 雙爪取盒
        END_CASE

{region '第一階段：從圓帶取盒'}
	//=====================================================================
	// 第一階段：從圓帶取盒 (Pick from RoundBelt)
	//=====================================================================

    10000: // A爪單爪 - 移動圓帶到目標站位 (照抄 V2 step 61000 模式)
		DAS_CoreSys.MachineControl.fbAllocateArea.M_GetRoundBeltAccess(ControlAccess := E_RoundBeltControlAccess.FanucRobot);
		DAS_CoreSys.MachineControl.fbAllocateArea.M_StartReloadRoundBeltAtion(ReloadStation := info.ClampA_Setting.RoundBeltSetting.Station);
		IF RoundBelt.xDone AND arAxisCtrl_gb[AxisNo.RoundBelt].Admin.Axis.Status.NotMoving THEN
			DAS_CoreSys.MachineControl.fbAllocateArea.M_ResetReloadRoundBeltAction();
			CarrierReady_1st := TRUE;
			uiExecutingStep := 10010;
		END_IF
		IF RoundBelt.xError THEN
			_Error := TRUE;
			DAS_CoreSys.MachineControl.fbAllocateArea.M_ResetReloadRoundBeltAction();
			strStatus := '';
		END_IF
	10010: // A爪從圓帶取盒 (使用 PickBoxFromRoundBelt，與 V2 MoveBoxToRoundBelt 對稱)
		IF NOT Robot._DI1.Done THEN
			Robot.M_StartPickBoxFromRoundBelt_ClampA(
				CarrierSelect := info.ClampA_Setting.RoundBeltSetting.ReloadCarrier,
				A2_Sensor     := A2_Sensor,
				A3_Sensor     := A3_Sensor,
				RoundBeltSafe := CarrierReady_1st);
			_AClampDoingWork := TRUE;
		ELSE
			tonTimeOut.IN := FALSE;
			uiExecutingStep := 10080;
		END_IF
		tonTimeOut.IN := TRUE;
		IF tonTimeOut.Q THEN
			uiResumeStep := 10010;
			_Abort := TRUE;
			tonTimeOut.IN := FALSE;
			strStatus := 'FB_FeedInRoundBeltBoxToWareHouse ,Step 10010: Robot Move TimeOut';
		END_IF
		IF Robot.Error THEN
			uiResumeStep := 10010;
			strStatus := CONCAT('FB_FeedInRoundBeltBoxToWareHouse ,Step 10010: ', Robot.ErrMsg);
			_Abort := TRUE;
		END_IF
    10080: // A爪取盒完成，釋放圓帶控制權，清除手臂命令，跳到放盒階段
		DAS_CoreSys.MachineControl.fbAllocateArea.M_ResetReloadRoundBeltAction();
		DAS_CoreSys.MachineControl.fbAllocateArea.M_ReleaseRoundBeltAccess(ControlAccess := E_RoundBeltControlAccess.FanucRobot);
        Robot.M_ResetAllCommand();
        IF NOT Robot._DI1.Done THEN
            uiExecutingStep := 60000; // 跳到 A爪放盒到倉儲
        END_IF

    20000: // B爪單爪 - 移動圓帶到目標站位 (照抄 V2 模式)
		DAS_CoreSys.MachineControl.fbAllocateArea.M_GetRoundBeltAccess(ControlAccess := E_RoundBeltControlAccess.FanucRobot);
		DAS_CoreSys.MachineControl.fbAllocateArea.M_StartReloadRoundBeltAtion(ReloadStation := info.ClampB_Setting.RoundBeltSetting.Station);
		IF RoundBelt.xDone AND arAxisCtrl_gb[AxisNo.RoundBelt].Admin.Axis.Status.NotMoving THEN
			DAS_CoreSys.MachineControl.fbAllocateArea.M_ResetReloadRoundBeltAction();
			CarrierReady_2nd := TRUE;
			uiExecutingStep := 20010;
		END_IF
		IF RoundBelt.xError THEN
			_Error := TRUE;
			DAS_CoreSys.MachineControl.fbAllocateArea.M_ResetReloadRoundBeltAction();
			strStatus := CONCAT('FB_FeedInRoundBeltBoxToWareHouse ,Step 20000: ',RoundBelt.ErrorMsg);
		END_IF
	20010: // B爪從圓帶取盒 (使用 PickBoxFromRoundBelt)
		IF NOT Robot._DI1.Done THEN
			Robot.M_StartPickBoxFromRoundBelt_ClampB(
				CarrierSelect := info.ClampB_Setting.RoundBeltSetting.ReloadCarrier,
				A2_Sensor     := A2_Sensor,
				A3_Sensor     := A3_Sensor,
				RoundBeltSafe := CarrierReady_2nd);
			_BClampDoingWork := TRUE;
		ELSE
			tonTimeOut.IN := FALSE;
			uiExecutingStep := 20080;
		END_IF
		tonTimeOut.IN := TRUE;
		IF tonTimeOut.Q THEN
			uiResumeStep := 20010;
			_Abort := TRUE;
			tonTimeOut.IN := FALSE;
			strStatus := 'FB_FeedInRoundBeltBoxToWareHouse ,Step 20010: Robot Move Timeout';
		END_IF
		IF Robot.Error THEN
			uiResumeStep := 20010;
			strStatus := CONCAT('FB_FeedInRoundBeltBoxToWareHouse ,Step 20010: ', Robot.ErrMsg);
			_Abort := TRUE;
		END_IF
    20080: // B爪取盒完成，釋放圓帶控制權，清除手臂命令，跳到放盒階段
		DAS_CoreSys.MachineControl.fbAllocateArea.M_ResetReloadRoundBeltAction();
		DAS_CoreSys.MachineControl.fbAllocateArea.M_ReleaseRoundBeltAccess(ControlAccess := E_RoundBeltControlAccess.FanucRobot);
        Robot.M_ResetAllCommand();
        IF NOT Robot._DI1.Done THEN
            uiExecutingStep := 70000; // 跳到 B爪放盒到倉儲
        END_IF

    30000: // 雙爪取盒 - 先移動圓帶到 A爪站位 (照抄 V2 模式)
		DAS_CoreSys.MachineControl.fbAllocateArea.M_GetRoundBeltAccess(ControlAccess := E_RoundBeltControlAccess.FanucRobot);
		DAS_CoreSys.MachineControl.fbAllocateArea.M_StartReloadRoundBeltAtion(ReloadStation := info.ClampA_Setting.RoundBeltSetting.Station);
		IF RoundBelt.xDone AND arAxisCtrl_gb[AxisNo.RoundBelt].Admin.Axis.Status.NotMoving THEN
			DAS_CoreSys.MachineControl.fbAllocateArea.M_ResetReloadRoundBeltAction();
			CarrierReady_1st := TRUE;
			uiExecutingStep := 30010;
		END_IF
		IF RoundBelt.xError THEN
			_Error := TRUE;
			DAS_CoreSys.MachineControl.fbAllocateArea.M_ResetReloadRoundBeltAction();
			strStatus := CONCAT('FB_FeedInRoundBeltBoxToWareHouse ,Step 30000: ',RoundBelt.ErrorMsg);
		END_IF
	30010: // 雙爪 A爪從圓帶取盒 (使用 PickBoxFromRoundBelt)
		IF NOT Robot._DI1.Done THEN
			Robot.M_StartPickBoxFromRoundBelt_ClampA(
				CarrierSelect := info.ClampA_Setting.RoundBeltSetting.ReloadCarrier,
				A2_Sensor     := A2_Sensor,
				A3_Sensor     := A3_Sensor,
				RoundBeltSafe := CarrierReady_1st);
			_AClampDoingWork := TRUE;
		ELSE
			tonTimeOut.IN := FALSE;
			uiExecutingStep := 30080;
		END_IF
		tonTimeOut.IN := TRUE;
		IF tonTimeOut.Q THEN
			uiResumeStep := 30010;
			_Abort := TRUE;
			tonTimeOut.IN := FALSE;
			strStatus := 'FB_FeedInRoundBeltBoxToWareHouse ,Step 30010 : Robot Move Timeout';
		END_IF
		IF Robot.Error THEN
			uiResumeStep := 30010;
			strStatus := CONCAT('FB_FeedInRoundBeltBoxToWareHouse ,Step 30010: ', Robot.ErrMsg);
			_Abort := TRUE;
		END_IF
	30080: // A爪取盒完成，清除手臂命令，準備 B爪取盒 (同站/不同站都重新移動圓帶)
		Robot.M_ResetAllCommand();
		IF NOT Robot._DI1.Done THEN
			uiExecutingStep := 31000;
		END_IF
	31000: // 移動圓帶到 B爪目標站位 (照抄 V2 模式)
		DAS_CoreSys.MachineControl.fbAllocateArea.M_GetRoundBeltAccess(ControlAccess := E_RoundBeltControlAccess.FanucRobot);
		DAS_CoreSys.MachineControl.fbAllocateArea.M_StartReloadRoundBeltAtion(ReloadStation := info.ClampB_Setting.RoundBeltSetting.Station);
		IF RoundBelt.xDone AND arAxisCtrl_gb[AxisNo.RoundBelt].Admin.Axis.Status.NotMoving THEN
			DAS_CoreSys.MachineControl.fbAllocateArea.M_ResetReloadRoundBeltAction();
			CarrierReady_2nd := TRUE;
			uiExecutingStep := 31010;
		END_IF
		IF RoundBelt.xError THEN
			_Error := TRUE;
			DAS_CoreSys.MachineControl.fbAllocateArea.M_ResetReloadRoundBeltAction();
			strStatus := CONCAT('FB_FeedInRoundBeltBoxToWareHouse ,Step 31000: ',RoundBelt.ErrorMsg);
		END_IF
	31010: // 雙爪 B爪從圓帶取盒 (使用 PickBoxFromRoundBelt)
		IF NOT Robot._DI1.Done THEN
			Robot.M_StartPickBoxFromRoundBelt_ClampB(
				CarrierSelect := info.ClampB_Setting.RoundBeltSetting.ReloadCarrier,
				A2_Sensor     := A2_Sensor,
				A3_Sensor     := A3_Sensor,
				RoundBeltSafe := CarrierReady_2nd);
			_BClampDoingWork := TRUE;
		ELSE
			tonTimeOut.IN := FALSE;
			uiExecutingStep := 31080;
		END_IF
		tonTimeOut.IN := TRUE;
		IF tonTimeOut.Q THEN
			uiResumeStep := 31010;
			_Abort := TRUE;
			tonTimeOut.IN := FALSE;
			strStatus := 'FB_FeedInRoundBeltBoxToWareHouse ,Step 31010 : Robot Move Timeout';
		END_IF
		IF Robot.Error THEN
			uiResumeStep := 31010;
			strStatus := CONCAT('FB_FeedInRoundBeltBoxToWareHouse ,Step 31010: ', Robot.ErrMsg);
			_Abort := TRUE;
		END_IF
	31080: // 雙爪取盒完成，釋放圓帶控制權，跳到放盒階段
		DAS_CoreSys.MachineControl.fbAllocateArea.M_ResetReloadRoundBeltAction();
		DAS_CoreSys.MachineControl.fbAllocateArea.M_ReleaseRoundBeltAccess(ControlAccess := E_RoundBeltControlAccess.FanucRobot);
		Robot.M_ResetAllCommand();
		IF NOT Robot._DI1.Done THEN
			uiExecutingStep := 80000; // 跳到雙爪放盒到倉儲
		END_IF
{endregion}

{region '第二階段：放盒到倉儲'}
	//=====================================================================
	// 第二階段：放盒到倉儲 (Place to WareHouse)
	//=====================================================================

    60000: // A爪單爪放盒 - 清除手臂命令，確認手臂閒置
        Robot.M_ResetAllCommand();
        // 確認手臂沒有在執行其他動作
        IF NOT Robot._di1.Done AND
            NOT (Robot._DI1.AbsMoveA OR
            Robot._DI1.AbsMoveB OR
            Robot._DI1.WarehouseA OR
            Robot._DI1.WarehouseB) THEN
            uiExecutingStep := 61000;
        END_IF
    61000: // A爪放盒到倉儲 (照抄 V2 模式：同時驅動倉儲 FeedIn + Robot Place，光電板 sensor 確認軌道空)
		ClampA_WareHouseCoordinates := info.ClampA_Setting.WareHouseSetting;
        IF NOT Robot._DI1.Done THEN
            IF info.ClampA_Setting.PlaceArea = E_FeedInToWareHouse_PlaceArea.WareHouseA THEN
				WareHouse.M_StartFeedInBox(WareHouseSelect := E_WareHouse.WareHouseA, WarehouseCoordinates := ClampA_WareHouseCoordinates);
				IF WareHouse.bFeedInBox_Completed THEN
					BoxReady_1st := TRUE;
				END_IF
                Robot.M_StartWareHousePlaceBox_ClampA(
                    WareHouseSelect := E_WareHouse.WareHouseA,
                    Info            := ClampA_WareHouseCoordinates,
                    BoxReady_1st    := BoxReady_1st);
            ELSIF info.ClampA_Setting.PlaceArea = E_FeedInToWareHouse_PlaceArea.WareHouseB THEN
				WareHouse.M_StartFeedInBox(WareHouseSelect := E_WareHouse.WareHouseB, WarehouseCoordinates := ClampA_WareHouseCoordinates);
				IF WareHouse.bFeedInBox_Completed THEN
					BoxReady_1st := TRUE;
				END_IF
                Robot.M_StartWareHousePlaceBox_ClampA(
                    WareHouseSelect := E_WareHouse.WareHouseB,
                    Info            := ClampA_WareHouseCoordinates,
                    BoxReady_1st    := BoxReady_1st);
            END_IF
        ELSE
			tonTimeOut.IN := FALSE;
            uiExecutingStep := 61080;
        END_IF
		tonTimeOut.IN := TRUE;
		IF tonTimeOut.Q THEN
			uiResumeStep := 61000;
			_Abort := TRUE;
			tonTimeOut.IN := FALSE;
			strStatus := 'FB_FeedInRoundBeltBoxToWareHouse ,Step 61000 : Robot Move Timeout';
		END_IF
    61080: // A爪放盒完成，設 AClampMoveDone，清除手臂命令
		AClampMoveDone := TRUE;
        Robot.M_ResetAllCommand();
        IF NOT Robot._DI1.Done THEN
            uiExecutingStep := 62000;
        END_IF
	62000: // 等待倉儲 FeedIn 完成 → Reset → 訊號關
		IF WareHouse.bFeedInBox_Completed THEN
			WareHouse.M_ResetFeedInBox();
			uiExecutingStep := 62010;
		END_IF
	62010:
		IF NOT WareHouse.bFeedInBox_Completed THEN
			uiExecutingStep := 99000;
		END_IF

    70000: // B爪單爪放盒 - 清除手臂命令，確認手臂閒置
        Robot.M_ResetAllCommand();
        IF NOT Robot._di1.Done AND
            NOT (Robot._DI1.AbsMoveA OR
            Robot._DI1.AbsMoveB OR
            Robot._DI1.WarehouseA OR
            Robot._DI1.WarehouseB) THEN
            uiExecutingStep := 71000;
        END_IF
    71000: // B爪放盒到倉儲 (照抄 V2 模式：同時驅動倉儲 FeedIn + Robot Place)
		ClampB_WareHouseCoordinates := info.ClampB_Setting.WareHouseSetting;
        IF NOT Robot._DI1.Done THEN
            IF info.ClampB_Setting.PlaceArea = E_FeedInToWareHouse_PlaceArea.WareHouseA THEN
				WareHouse.M_StartFeedInBox(WareHouseSelect := E_WareHouse.WareHouseA, WarehouseCoordinates := ClampB_WareHouseCoordinates);
				IF WareHouse.bFeedInBox_Completed THEN
					BoxReady_2nd := TRUE;
				END_IF
                Robot.M_StartWareHousePlaceBox_ClampB(
                    WareHouseSelect := E_WareHouse.WareHouseA,
                    Info            := ClampB_WareHouseCoordinates,
                    BoxReady_2nd    := BoxReady_2nd);
            ELSIF info.ClampB_Setting.PlaceArea = E_FeedInToWareHouse_PlaceArea.WareHouseB THEN
				WareHouse.M_StartFeedInBox(WareHouseSelect := E_WareHouse.WareHouseB, WarehouseCoordinates := ClampB_WareHouseCoordinates);
				IF WareHouse.bFeedInBox_Completed THEN
					BoxReady_2nd := TRUE;
				END_IF
                Robot.M_StartWareHousePlaceBox_ClampB(
                    WareHouseSelect := E_WareHouse.WareHouseB,
                    Info            := ClampB_WareHouseCoordinates,
                    BoxReady_2nd    := BoxReady_2nd);
            END_IF
        ELSE
			tonTimeOut.IN := FALSE;
            uiExecutingStep := 71080;
        END_IF
		tonTimeOut.IN := TRUE;
		IF tonTimeOut.Q THEN
			uiResumeStep := 71000;
			_Abort := TRUE;
			tonTimeOut.IN := FALSE;
			strStatus := 'FB_FeedInRoundBeltBoxToWareHouse ,Step 71000 : Robot Move Timeout';
		END_IF
    71080: // B爪放盒完成，設 BClampMoveDone，清除手臂命令
		BClampMoveDone := TRUE;
        Robot.M_ResetAllCommand();
        IF NOT Robot._DI1.Done THEN
            uiExecutingStep := 72000;
        END_IF
	72000: // 等待倉儲 FeedIn 完成 → Reset → 訊號關
		IF WareHouse.bFeedInBox_Completed THEN
			WareHouse.M_ResetFeedInBox();
			uiExecutingStep := 72010;
		END_IF
	72010:
		IF NOT WareHouse.bFeedInBox_Completed THEN
			uiExecutingStep := 99000;
		END_IF

